ACTION CP03:
{region "CP03柜"}									
DI_[8,1](	ON:= , 	OFF:= , 	LINK:=EL1008[8,1] , 	VALUE=> 	arDropCylinder[11].i.InSensor	);	(*	料仓11气缸原位	*)
DI_[8,2](	ON:= , 	OFF:= , 	LINK:=EL1008[8,2] , 	VALUE=> 	arDropCylinder[11].i.OutSensor	);	(*	料仓11气缸工作位	*)
DI_[8,3](	ON:= , 	OFF:= , 	LINK:=EL1008[8,3] , 	VALUE=> 	arHighSensor[11].i.Link	);	(*	料仓11少料	*)
DI_[8,4](	ON:= , 	OFF:= , 	LINK:=EL1008[8,4] , 	VALUE=> 	arLowSensor[11].i.Link	);	(*	料仓11缺料	*)
DI_[8,5](	ON:= , 	OFF:= , 	LINK:=EL1008[8,5] , 	VALUE=> 	arDropCylinder[12].i.InSensor	);	(*	料仓12气缸原位	*)
DI_[8,6](	ON:= , 	OFF:= , 	LINK:=EL1008[8,6] , 	VALUE=> 	arDropCylinder[12].i.OutSensor	);	(*	料仓12气缸工作位	*)
DI_[8,7](	ON:= , 	OFF:= , 	LINK:=EL1008[8,7] , 	VALUE=> 	arHighSensor[12].i.Link	);	(*	料仓12少料	*)
DI_[8,8](	ON:= , 	OFF:= , 	LINK:=EL1008[8,8] , 	VALUE=> 	arLowSensor[12].i.Link	);	(*	料仓12缺料	*)
DI_[9,1](	ON:= , 	OFF:= , 	LINK:=EL1008[9,1] , 	VALUE=> 	arDropCylinder[13].i.InSensor	);	(*	料仓13气缸原位	*)
DI_[9,2](	ON:= , 	OFF:= , 	LINK:=EL1008[9,2] , 	VALUE=> 	arDropCylinder[13].i.OutSensor	);	(*	料仓13气缸工作位	*)
DI_[9,3](	ON:= , 	OFF:= , 	LINK:=EL1008[9,3] , 	VALUE=> 	arHighSensor[13].i.Link	);	(*	料仓13少料	*)
DI_[9,4](	ON:= , 	OFF:= , 	LINK:=EL1008[9,4] , 	VALUE=> 	arLowSensor[13].i.Link	);	(*	料仓13缺料	*)
DI_[9,5](	ON:= , 	OFF:= , 	LINK:=EL1008[9,5] , 	VALUE=> 	arDropCylinder[14].i.InSensor	);	(*	料仓14气缸原位	*)
DI_[9,6](	ON:= , 	OFF:= , 	LINK:=EL1008[9,6] , 	VALUE=> 	arDropCylinder[14].i.OutSensor	);	(*	料仓14气缸工作位	*)
DI_[9,7](	ON:= , 	OFF:= , 	LINK:=EL1008[9,7] , 	VALUE=> 	arHighSensor[14].i.Link	);	(*	料仓14少料	*)
DI_[9,8](	ON:= , 	OFF:= , 	LINK:=EL1008[9,8] , 	VALUE=> 	arLowSensor[14].i.Link	);	(*	料仓14缺料	*)
DI_[10,1](	ON:= , 	OFF:= , 	LINK:=EL1008[10,1] , 	VALUE=> 	arDropCylinder[15].i.InSensor	);	(*	料仓15气缸原位	*)
DI_[10,2](	ON:= , 	OFF:= , 	LINK:=EL1008[10,2] , 	VALUE=> 	arDropCylinder[15].i.OutSensor	);	(*	料仓15气缸工作位	*)
DI_[10,3](	ON:= , 	OFF:= , 	LINK:=EL1008[10,3] , 	VALUE=> 	arHighSensor[15].i.Link	);	(*	料仓15少料	*)
DI_[10,4](	ON:= , 	OFF:= , 	LINK:=EL1008[10,4] , 	VALUE=> 	arLowSensor[15].i.Link	);	(*	料仓15缺料	*)
DI_[10,5](	ON:= , 	OFF:= , 	LINK:=EL1008[10,5] , 	VALUE=> 	arDropCylinder[16].i.InSensor	);	(*	料仓16气缸原位	*)
DI_[10,6](	ON:= , 	OFF:= , 	LINK:=EL1008[10,6] , 	VALUE=> 	arDropCylinder[16].i.OutSensor	);	(*	料仓16气缸工作位	*)
DI_[10,7](	ON:= , 	OFF:= , 	LINK:=EL1008[10,7] , 	VALUE=> 	arHighSensor[16].i.Link	);	(*	料仓16少料	*)
DI_[10,8](	ON:= , 	OFF:= , 	LINK:=EL1008[10,8] , 	VALUE=> 	arLowSensor[16].i.Link	);	(*	料仓16缺料	*)
DI_[11,1](	ON:= , 	OFF:= , 	LINK:=EL1008[11,1] , 	VALUE=> 	arDropCylinder[17].i.InSensor	);	(*	料仓17气缸原位	*)
DI_[11,2](	ON:= , 	OFF:= , 	LINK:=EL1008[11,2] , 	VALUE=> 	arDropCylinder[17].i.OutSensor	);	(*	料仓17气缸工作位	*)
DI_[11,3](	ON:= , 	OFF:= , 	LINK:=EL1008[11,3] , 	VALUE=> 	arHighSensor[17].i.Link	);	(*	料仓17少料	*)
DI_[11,4](	ON:= , 	OFF:= , 	LINK:=EL1008[11,4] , 	VALUE=> 	arLowSensor[17].i.Link	);	(*	料仓17缺料	*)
DI_[11,5](	ON:= , 	OFF:= , 	LINK:=EL1008[11,5] , 	VALUE=> 	arDropCylinder[18].i.InSensor	);	(*	料仓18气缸原位	*)
DI_[11,6](	ON:= , 	OFF:= , 	LINK:=EL1008[11,6] , 	VALUE=> 	arDropCylinder[18].i.OutSensor	);	(*	料仓18气缸工作位	*)
DI_[11,7](	ON:= , 	OFF:= , 	LINK:=EL1008[11,7] , 	VALUE=> 	arHighSensor[18].i.Link	);	(*	料仓18少料	*)
DI_[11,8](	ON:= , 	OFF:= , 	LINK:=EL1008[11,8] , 	VALUE=> 	arLowSensor[18].i.Link	);	(*	料仓18缺料	*)
DI_[12,1](	ON:= , 	OFF:= , 	LINK:=EL1008[12,1] , 	VALUE=> 	arDropCylinder[19].i.InSensor	);	(*	料仓19气缸原位	*)
DI_[12,2](	ON:= , 	OFF:= , 	LINK:=EL1008[12,2] , 	VALUE=> 	arDropCylinder[19].i.OutSensor	);	(*	料仓19气缸工作位	*)
DI_[12,3](	ON:= , 	OFF:= , 	LINK:=EL1008[12,3] , 	VALUE=> 	arHighSensor[19].i.Link	);	(*	料仓19少料	*)
DI_[12,4](	ON:= , 	OFF:= , 	LINK:=EL1008[12,4] , 	VALUE=> 	arLowSensor[19].i.Link	);	(*	料仓19缺料	*)
DI_[12,5](	ON:= , 	OFF:= , 	LINK:=EL1008[12,5] , 	VALUE=> 	arDropCylinder[20].i.InSensor	);	(*	料仓20气缸原位	*)
DI_[12,6](	ON:= , 	OFF:= , 	LINK:=EL1008[12,6] , 	VALUE=> 	arDropCylinder[20].i.OutSensor	);	(*	料仓20气缸工作位	*)
DI_[12,7](	ON:= , 	OFF:= , 	LINK:=EL1008[12,7] , 	VALUE=> 	arHighSensor[20].i.Link	);	(*	料仓20少料	*)
DI_[12,8](	ON:= , 	OFF:= , 	LINK:=EL1008[12,8] , 	VALUE=> 	arLowSensor[20].i.Link	);	(*	料仓20缺料	*)		
DI_[13,1](	ON:= , 	OFF:= , 	LINK:=EL1008[13,1] , 	VALUE=> 	arDropSensor[11].i.Link	);	(*	工位11落料	*)
DI_[13,2](	ON:= , 	OFF:= , 	LINK:=EL1008[13,2] , 	VALUE=> 	arDropSensor[12].i.Link	);	(*	工位12落料	*)
DI_[13,3](	ON:= , 	OFF:= , 	LINK:=EL1008[13,3] , 	VALUE=> 	arDropSensor[13].i.Link	);	(*	工位13落料	*)
DI_[13,4](	ON:= , 	OFF:= , 	LINK:=EL1008[13,4] , 	VALUE=> 	arDropSensor[14].i.Link	);	(*	工位14落料	*)
DI_[13,5](	ON:= , 	OFF:= , 	LINK:=EL1008[13,5] , 	VALUE=> 	arDropSensor[15].i.Link	);	(*	工位15落料	*)
DI_[13,6](	ON:= , 	OFF:= , 	LINK:=EL1008[13,6] , 	VALUE=> 	arDropSensor[16].i.Link	);	(*	工位16落料	*)
DI_[13,7](	ON:= , 	OFF:= , 	LINK:=EL1008[13,7] , 	VALUE=> 	arDropSensor[17].i.Link	);	(*	工位17落料	*)
DI_[13,8](	ON:= , 	OFF:= , 	LINK:=EL1008[13,8] , 	VALUE=> 	arDropSensor[18].i.Link	);	(*	工位18落料	*)
DI_[14,1](	ON:= , 	OFF:= , 	LINK:=EL1008[14,1] , 	VALUE=> 	arDropSensor[19].i.Link	);	(*	工位19落料	*)
DI_[14,2](	ON:= , 	OFF:= , 	LINK:=EL1008[14,2] , 	VALUE=> 	arDropSensor[20].i.Link	);	(*	工位20落料	*)
DI_[14,3](	ON:= , 	OFF:= , 	LINK:=EL1008[14,3] , 	VALUE=> 	arSafeDoorSts[5]	);	(*	安全门5	*)
DI_[14,4](	ON:= , 	OFF:= , 	LINK:=EL1008[14,4] , 	VALUE=> 	arSafeDoorSts[6]	);	(*	安全门6	*)
DI_[14,5](	ON:= , 	OFF:= , 	LINK:=EL1008[14,5] , 	VALUE=> 	arSafeDoorSts[7]	);	(*	安全门7	*)
DI_[14,6](	ON:= , 	OFF:= , 	LINK:=EL1008[14,6] , 	VALUE=> 	arSafeDoorSts[8]	);	(*	安全门8	*)
DI_[14,7](	ON:= , 	OFF:= , 	LINK:=EL1008[14,7] , 	VALUE=> 	arSafeDoorSts[9]	);	(*	安全门9	*)
DI_[14,8](	ON:= , 	OFF:= , 	LINK:=EL1008[14,8] , 	VALUE=> 	glb_bAirFeedback_UN01[2]	);	(*	数粒系统气压反馈	*)
DI_[30,1](	ON:= , 	OFF:= , 	LINK:=EL1008[30,1] , 	VALUE=> 	arDropBufferCyclinder[1].i.InSensor	);	(*	备用	*)
DI_[30,2](	ON:= , 	OFF:= , 	LINK:=EL1008[30,2] , 	VALUE=> 		);	(*	备用	*)
DI_[30,3](	ON:= , 	OFF:= , 	LINK:=EL1008[30,3] , 	VALUE=> 		);	(*	备用	*)
DI_[30,4](	ON:= , 	OFF:= , 	LINK:=EL1008[30,4] , 	VALUE=> 		);	(*	备用	*)
DI_[30,5](	ON:= , 	OFF:= , 	LINK:=EL1008[30,5] , 	VALUE=> 		);	(*	备用	*)
DI_[30,6](	ON:= , 	OFF:= , 	LINK:=EL1008[30,6] , 	VALUE=> 		);	(*	备用	*)
DI_[30,7](	ON:= , 	OFF:= , 	LINK:=EL1008[30,7] , 	VALUE=> 		);	(*	备用	*)
DI_[30,8](	ON:= , 	OFF:= , 	LINK:=EL1008[30,8] , 	VALUE=> 		);	(*	备用	*)


arDropBufferCyclinder[1].i.OutSensor:= NOT arDropBufferCyclinder[1].i.InSensor;
arDropBufferCyclinder[2].i.OutSensor:= NOT arDropBufferCyclinder[2].i.InSensor;		  
(*****************************************************************************************************)									
DO_[8,1](	ON:= , 	OFF:= , 	LINK=>EL2008[8,1] , 	VALUE:= 	arDropCylinder[11].o.ValveIn	);	(*	料仓11气缸原位	*)
DO_[8,2](	ON:= , 	OFF:= , 	LINK=>EL2008[8,2] , 	VALUE:= 	arDropCylinder[11].o.ValveOut	);	(*	料仓11气缸工作位	*)
DO_[8,3](	ON:= , 	OFF:= , 	LINK=>EL2008[8,3] , 	VALUE:= 	arDropCylinder[12].o.ValveIn	);	(*	料仓12气缸原位	*)
DO_[8,4](	ON:= , 	OFF:= , 	LINK=>EL2008[8,4] , 	VALUE:= 	arDropCylinder[12].o.ValveOut	);	(*	料仓12气缸工作位	*)
DO_[8,5](	ON:= , 	OFF:= , 	LINK=>EL2008[8,5] , 	VALUE:= 	arDropCylinder[13].o.ValveIn	);	(*	料仓13气缸原位	*)
DO_[8,6](	ON:= , 	OFF:= , 	LINK=>EL2008[8,6] , 	VALUE:= 	arDropCylinder[13].o.ValveOut	);	(*	料仓13气缸工作位	*)
DO_[8,7](	ON:= , 	OFF:= , 	LINK=>EL2008[8,7] , 	VALUE:= 	arDropCylinder[14].o.ValveIn	);	(*	料仓14气缸原位	*)
DO_[8,8](	ON:= , 	OFF:= , 	LINK=>EL2008[8,8] , 	VALUE:= 	arDropCylinder[14].o.ValveOut	);	(*	料仓14气缸工作位	*)
DO_[9,1](	ON:= , 	OFF:= , 	LINK=>EL2008[9,1] , 	VALUE:= 	arDropCylinder[15].o.ValveIn	);	(*	料仓15气缸原位	*)
DO_[9,2](	ON:= , 	OFF:= , 	LINK=>EL2008[9,2] , 	VALUE:= 	arDropCylinder[15].o.ValveOut	);	(*	料仓15气缸工作位	*)
DO_[9,3](	ON:= , 	OFF:= , 	LINK=>EL2008[9,3] , 	VALUE:= 	arDropCylinder[16].o.ValveIn	);	(*	料仓16气缸原位	*)
DO_[9,4](	ON:= , 	OFF:= , 	LINK=>EL2008[9,4] , 	VALUE:= 	arDropCylinder[16].o.ValveOut	);	(*	料仓16气缸工作位	*)
DO_[9,5](	ON:= , 	OFF:= , 	LINK=>EL2008[9,5] , 	VALUE:= 	arDropCylinder[17].o.ValveIn	);	(*	料仓17气缸原位	*)
DO_[9,6](	ON:= , 	OFF:= , 	LINK=>EL2008[9,6] , 	VALUE:= 	arDropCylinder[17].o.ValveOut	);	(*	料仓17气缸工作位	*)
DO_[9,7](	ON:= , 	OFF:= , 	LINK=>EL2008[9,7] , 	VALUE:= 	arDropCylinder[18].o.ValveIn	);	(*	料仓18气缸原位	*)
DO_[9,8](	ON:= , 	OFF:= , 	LINK=>EL2008[9,8] , 	VALUE:= 	arDropCylinder[18].o.ValveOut	);	(*	料仓18气缸工作位	*)
DO_[10,1](	ON:= , 	OFF:= , 	LINK=>EL2008[10,1] , 	VALUE:= 	arDropCylinder[19].o.ValveIn	);	(*	料仓19气缸原位	*)
DO_[10,2](	ON:= , 	OFF:= , 	LINK=>EL2008[10,2] , 	VALUE:= 	arDropCylinder[19].o.ValveOut	);	(*	料仓19气缸工作位	*)
DO_[10,3](	ON:= , 	OFF:= , 	LINK=>EL2008[10,3] , 	VALUE:= 	arDropCylinder[20].o.ValveIn	);	(*	料仓20气缸原位	*)
DO_[10,4](	ON:= , 	OFF:= , 	LINK=>EL2008[10,4] , 	VALUE:= 	arDropCylinder[20].o.ValveOut	);	(*	料仓20气缸工作位	*)
DO_[10,5](	ON:= , 	OFF:= , 	LINK=>EL2008[10,5] , 	VALUE:= 	arCounters[11].LineVibrator_Wrk	);	(*	料仓11直震启动	*)
DO_[10,6](	ON:= , 	OFF:= , 	LINK=>EL2008[10,6] , 	VALUE:= 	arCounters[11].CircleVibrator_Wrk	);	(*	料仓11圆震启动	*)
DO_[10,7](	ON:= , 	OFF:= , 	LINK=>EL2008[10,7] , 	VALUE:= 	arCounters[11].DropVibrator_Wrk	);	(*	料仓11落料启动	*)
DO_[10,8](	ON:= , 	OFF:= , 	LINK=>EL2008[10,8] , 	VALUE:= 	arCounters[12].LineVibrator_Wrk	);	(*	料仓12直震启动	*)
DO_[11,1](	ON:= , 	OFF:= , 	LINK=>EL2008[11,1] , 	VALUE:= 	arCounters[12].CircleVibrator_Wrk	);	(*	料仓12圆震启动	*)
DO_[11,2](	ON:= , 	OFF:= , 	LINK=>EL2008[11,2] , 	VALUE:= 	arCounters[12].DropVibrator_Wrk	);	(*	料仓12落料启动	*)
DO_[11,3](	ON:= , 	OFF:= , 	LINK=>EL2008[11,3] , 	VALUE:= 	arCounters[13].LineVibrator_Wrk	);	(*	料仓13直震启动	*)
DO_[11,4](	ON:= , 	OFF:= , 	LINK=>EL2008[11,4] , 	VALUE:= 	arCounters[13].CircleVibrator_Wrk	);	(*	料仓13圆震启动	*)
DO_[11,5](	ON:= , 	OFF:= , 	LINK=>EL2008[11,5] , 	VALUE:= 	arCounters[13].DropVibrator_Wrk	);	(*	料仓13落料启动	*)
DO_[11,6](	ON:= , 	OFF:= , 	LINK=>EL2008[11,6] , 	VALUE:= 	arCounters[14].LineVibrator_Wrk	);	(*	料仓14直震启动	*)
DO_[11,7](	ON:= , 	OFF:= , 	LINK=>EL2008[11,7] , 	VALUE:= 	arCounters[14].CircleVibrator_Wrk	);	(*	料仓14圆震启动	*)
DO_[11,8](	ON:= , 	OFF:= , 	LINK=>EL2008[11,8] , 	VALUE:= 	arCounters[14].DropVibrator_Wrk	);	(*	料仓14落料启动	*)
DO_[12,1](	ON:= , 	OFF:= , 	LINK=>EL2008[12,1] , 	VALUE:= 	arCounters[15].LineVibrator_Wrk	);	(*	料仓15直震启动	*)
DO_[12,2](	ON:= , 	OFF:= , 	LINK=>EL2008[12,2] , 	VALUE:= 	arCounters[15].CircleVibrator_Wrk	);	(*	料仓15圆震启动	*)
DO_[12,3](	ON:= , 	OFF:= , 	LINK=>EL2008[12,3] , 	VALUE:= 	arCounters[15].DropVibrator_Wrk	);	(*	料仓15落料启动	*)
DO_[12,4](	ON:= , 	OFF:= , 	LINK=>EL2008[12,4] , 	VALUE:= 	arCounters[16].LineVibrator_Wrk	);	(*	料仓16直震启动	*)
DO_[12,5](	ON:= , 	OFF:= , 	LINK=>EL2008[12,5] , 	VALUE:= 	arCounters[16].CircleVibrator_Wrk	);	(*	料仓16圆震启动	*)
DO_[12,6](	ON:= , 	OFF:= , 	LINK=>EL2008[12,6] , 	VALUE:= 	arCounters[16].DropVibrator_Wrk	);	(*	料仓16落料启动	*)
DO_[12,7](	ON:= , 	OFF:= , 	LINK=>EL2008[12,7] , 	VALUE:= 	arCounters[17].LineVibrator_Wrk	);	(*	料仓17直震启动	*)
DO_[12,8](	ON:= , 	OFF:= , 	LINK=>EL2008[12,8] , 	VALUE:= 	arCounters[17].CircleVibrator_Wrk	);	(*	料仓17圆震启动	*)
DO_[13,1](	ON:= , 	OFF:= , 	LINK=>EL2008[13,1] , 	VALUE:= 	arCounters[17].DropVibrator_Wrk	);	(*	料仓17落料启动	*)
DO_[13,2](	ON:= , 	OFF:= , 	LINK=>EL2008[13,2] , 	VALUE:= 	arCounters[18].LineVibrator_Wrk	);	(*	料仓18直震启动	*)
DO_[13,3](	ON:= , 	OFF:= , 	LINK=>EL2008[13,3] , 	VALUE:= 	arCounters[18].CircleVibrator_Wrk	);	(*	料仓18圆震启动	*)
DO_[13,4](	ON:= , 	OFF:= , 	LINK=>EL2008[13,4] , 	VALUE:= 	arCounters[18].DropVibrator_Wrk	);	(*	料仓18落料启动	*)
DO_[13,5](	ON:= , 	OFF:= , 	LINK=>EL2008[13,5] , 	VALUE:= 	arCounters[19].LineVibrator_Wrk	);	(*	料仓19直震启动	*)
DO_[13,6](	ON:= , 	OFF:= , 	LINK=>EL2008[13,6] , 	VALUE:= 	arCounters[19].CircleVibrator_Wrk	);	(*	料仓19圆震启动	*)
DO_[13,7](	ON:= , 	OFF:= , 	LINK=>EL2008[13,7] , 	VALUE:= 	arCounters[19].DropVibrator_Wrk	);	(*	料仓19落料启动	*)
DO_[13,8](	ON:= , 	OFF:= , 	LINK=>EL2008[13,8] , 	VALUE:= 	arCounters[20].LineVibrator_Wrk	);	(*	料仓20直震启动	*)
DO_[14,1](	ON:= , 	OFF:= , 	LINK=>EL2008[14,1] , 	VALUE:= 	arCounters[20].CircleVibrator_Wrk	);	(*	料仓20圆震启动	*)
DO_[14,2](	ON:= , 	OFF:= , 	LINK=>EL2008[14,2] , 	VALUE:= 	arCounters[20].DropVibrator_Wrk	);	(*	料仓20落料启动	*)
DO_[14,3](	ON:= , 	OFF:= , 	LINK=>EL2008[14,3] , 	VALUE:= 	glb_arLightRelay_UN01[1]	);	(*设备照明灯继电器1	*)
DO_[14,4](	ON:= , 	OFF:= , 	LINK=>EL2008[14,4] , 	VALUE:= 	glb_bCounterAirValve_UN01	);	(*数粒系统气压阀	*)
DO_[14,5](	ON:= , 	OFF:= , 	LINK=>EL2008[14,5] , 	VALUE:=     arDropBufferCyclinder[1].o.ValveOut);	(**)
DO_[14,6](	ON:= , 	OFF:= , 	LINK=>EL2008[14,6] , 	VALUE:= 	arDropBufferCyclinder[2].o.ValveOut);	(**)
DO_[14,7](	ON:= , 	OFF:= , 	LINK=>EL2008[14,7] , 	VALUE:= 	);	(**)
DO_[14,8](	ON:= , 	OFF:= , 	LINK=>EL2008[14,8] , 	VALUE:= 	);	(**)									
{endregion}
END_ACTION

ACTION CP04:
{region "CP04柜"}									
DI_[15,1](	ON:= , 	OFF:= , 	LINK:=EL1008[15,1] , 	VALUE=> 	arDropCylinder[21].i.InSensor	);	(*	料仓21气缸原位	*)
DI_[15,2](	ON:= , 	OFF:= , 	LINK:=EL1008[15,2] , 	VALUE=> 	arDropCylinder[21].i.OutSensor	);	(*	料仓21气缸工作位	*)
DI_[15,3](	ON:= , 	OFF:= , 	LINK:=EL1008[15,3] , 	VALUE=> 	arHighSensor[21].i.Link	);	(*	料仓21少料	*)
DI_[15,4](	ON:= , 	OFF:= , 	LINK:=EL1008[15,4] , 	VALUE=> 	arLowSensor[21].i.Link	);	(*	料仓21缺料	*)
DI_[15,5](	ON:= , 	OFF:= , 	LINK:=EL1008[15,5] , 	VALUE=> 	arDropCylinder[22].i.InSensor	);	(*	料仓22气缸原位	*)
DI_[15,6](	ON:= , 	OFF:= , 	LINK:=EL1008[15,6] , 	VALUE=> 	arDropCylinder[22].i.OutSensor	);	(*	料仓22气缸工作位	*)
DI_[15,7](	ON:= , 	OFF:= , 	LINK:=EL1008[15,7] , 	VALUE=> 	arHighSensor[22].i.Link	);	(*	料仓22少料	*)
DI_[15,8](	ON:= , 	OFF:= , 	LINK:=EL1008[15,8] , 	VALUE=> 	arLowSensor[22].i.Link	);	(*	料仓22缺料	*)
DI_[16,1](	ON:= , 	OFF:= , 	LINK:=EL1008[16,1] , 	VALUE=> 	arDropCylinder[23].i.InSensor	);	(*	料仓23气缸原位	*)
DI_[16,2](	ON:= , 	OFF:= , 	LINK:=EL1008[16,2] , 	VALUE=> 	arDropCylinder[23].i.OutSensor	);	(*	料仓23气缸工作位	*)
DI_[16,3](	ON:= , 	OFF:= , 	LINK:=EL1008[16,3] , 	VALUE=> 	arHighSensor[23].i.Link	);	(*	料仓23少料	*)
DI_[16,4](	ON:= , 	OFF:= , 	LINK:=EL1008[16,4] , 	VALUE=> 	arLowSensor[23].i.Link	);	(*	料仓23缺料	*)
DI_[16,5](	ON:= , 	OFF:= , 	LINK:=EL1008[16,5] , 	VALUE=> 	arDropCylinder[24].i.InSensor	);	(*	料仓24气缸原位	*)
DI_[16,6](	ON:= , 	OFF:= , 	LINK:=EL1008[16,6] , 	VALUE=> 	arDropCylinder[24].i.OutSensor	);	(*	料仓24气缸工作位	*)
DI_[16,7](	ON:= , 	OFF:= , 	LINK:=EL1008[16,7] , 	VALUE=> 	arHighSensor[24].i.Link	);	(*	料仓24少料	*)
DI_[16,8](	ON:= , 	OFF:= , 	LINK:=EL1008[16,8] , 	VALUE=> 	arLowSensor[24].i.Link	);	(*	料仓24缺料	*)
DI_[17,1](	ON:= , 	OFF:= , 	LINK:=EL1008[17,1] , 	VALUE=> 	arDropCylinder[25].i.InSensor	);	(*	料仓25气缸原位	*)
DI_[17,2](	ON:= , 	OFF:= , 	LINK:=EL1008[17,2] , 	VALUE=> 	arDropCylinder[25].i.OutSensor	);	(*	料仓25气缸工作位	*)
DI_[17,3](	ON:= , 	OFF:= , 	LINK:=EL1008[17,3] , 	VALUE=> 	arHighSensor[25].i.Link	);	(*	料仓25少料	*)
DI_[17,4](	ON:= , 	OFF:= , 	LINK:=EL1008[17,4] , 	VALUE=> 	arLowSensor[25].i.Link	);	(*	料仓25缺料	*)
DI_[17,5](	ON:= , 	OFF:= , 	LINK:=EL1008[17,5] , 	VALUE=> 	arDropCylinder[26].i.InSensor	);	(*	料仓26气缸原位	*)
DI_[17,6](	ON:= , 	OFF:= , 	LINK:=EL1008[17,6] , 	VALUE=> 	arDropCylinder[26].i.OutSensor	);	(*	料仓26气缸工作位	*)
DI_[17,7](	ON:= , 	OFF:= , 	LINK:=EL1008[17,7] , 	VALUE=> 	arHighSensor[26].i.Link	);	(*	料仓26少料	*)
DI_[17,8](	ON:= , 	OFF:= , 	LINK:=EL1008[17,8] , 	VALUE=> 	arLowSensor[26].i.Link	);	(*	料仓26缺料	*)
DI_[18,1](	ON:= , 	OFF:= , 	LINK:=EL1008[18,1] , 	VALUE=> 	arDropCylinder[27].i.InSensor	);	(*	料仓27气缸原位	*)
DI_[18,2](	ON:= , 	OFF:= , 	LINK:=EL1008[18,2] , 	VALUE=> 	arDropCylinder[27].i.OutSensor	);	(*	料仓27气缸工作位	*)
DI_[18,3](	ON:= , 	OFF:= , 	LINK:=EL1008[18,3] , 	VALUE=> 	arHighSensor[27].i.Link	);	(*	料仓27少料	*)
DI_[18,4](	ON:= , 	OFF:= , 	LINK:=EL1008[18,4] , 	VALUE=> 	arLowSensor[27].i.Link	);	(*	料仓27缺料	*)
DI_[18,5](	ON:= , 	OFF:= , 	LINK:=EL1008[18,5] , 	VALUE=> 	arDropCylinder[28].i.InSensor	);	(*	料仓28气缸原位	*)
DI_[18,6](	ON:= , 	OFF:= , 	LINK:=EL1008[18,6] , 	VALUE=> 	arDropCylinder[28].i.OutSensor	);	(*	料仓28气缸工作位	*)
DI_[18,7](	ON:= , 	OFF:= , 	LINK:=EL1008[18,7] , 	VALUE=> 	arHighSensor[28].i.Link	);	(*	料仓28少料	*)
DI_[18,8](	ON:= , 	OFF:= , 	LINK:=EL1008[18,8] , 	VALUE=> 	arLowSensor[28].i.Link	);	(*	料仓28缺料	*)
DI_[19,1](	ON:= , 	OFF:= , 	LINK:=EL1008[19,1] , 	VALUE=> 	arDropCylinder[29].i.InSensor	);	(*	料仓29气缸原位	*)
DI_[19,2](	ON:= , 	OFF:= , 	LINK:=EL1008[19,2] , 	VALUE=> 	arDropCylinder[29].i.OutSensor	);	(*	料仓29气缸工作位	*)
DI_[19,3](	ON:= , 	OFF:= , 	LINK:=EL1008[19,3] , 	VALUE=> 	arHighSensor[29].i.Link	);	(*	料仓29少料	*)
DI_[19,4](	ON:= , 	OFF:= , 	LINK:=EL1008[19,4] , 	VALUE=> 	arLowSensor[29].i.Link	);	(*	料仓29缺料	*)
DI_[19,5](	ON:= , 	OFF:= , 	LINK:=EL1008[19,5] , 	VALUE=> 	arDropCylinder[30].i.InSensor	);	(*	料仓30气缸原位	*)
DI_[19,6](	ON:= , 	OFF:= , 	LINK:=EL1008[19,6] , 	VALUE=> 	arDropCylinder[30].i.OutSensor	);	(*	料仓30气缸工作位	*)
DI_[19,7](	ON:= , 	OFF:= , 	LINK:=EL1008[19,7] , 	VALUE=> 	arHighSensor[30].i.Link	);	(*	料仓30少料	*)
DI_[19,8](	ON:= , 	OFF:= , 	LINK:=EL1008[19,8] , 	VALUE=> 	arLowSensor[30].i.Link	);	(*	料仓30缺料	*)
DI_[20,1](	ON:= , 	OFF:= , 	LINK:=EL1008[20,1] , 	VALUE=> 	arDropSensor[21].i.Link	);	(*	工位21落料	*)
DI_[20,2](	ON:= , 	OFF:= , 	LINK:=EL1008[20,2] , 	VALUE=> 	arDropSensor[22].i.Link	);	(*	工位22落料	*)
DI_[20,3](	ON:= , 	OFF:= , 	LINK:=EL1008[20,3] , 	VALUE=> 	arDropSensor[23].i.Link	);	(*	工位23落料	*)
DI_[20,4](	ON:= , 	OFF:= , 	LINK:=EL1008[20,4] , 	VALUE=> 	arDropSensor[24].i.Link	);	(*	工位24落料	*)
DI_[20,5](	ON:= , 	OFF:= , 	LINK:=EL1008[20,5] , 	VALUE=> 	arDropSensor[25].i.Link	);	(*	工位25落料	*)
DI_[20,6](	ON:= , 	OFF:= , 	LINK:=EL1008[20,6] , 	VALUE=> 	arDropSensor[26].i.Link	);	(*	工位26落料	*)
DI_[20,7](	ON:= , 	OFF:= , 	LINK:=EL1008[20,7] , 	VALUE=> 	arDropSensor[27].i.Link	);	(*	工位27落料	*)
DI_[20,8](	ON:= , 	OFF:= , 	LINK:=EL1008[20,8] , 	VALUE=> 	arDropSensor[28].i.Link	);	(*	工位28落料	*)
DI_[21,1](	ON:= , 	OFF:= , 	LINK:=EL1008[21,1] , 	VALUE=> 	arDropSensor[29].i.Link	);	(*	工位29落料	*)
DI_[21,2](	ON:= , 	OFF:= , 	LINK:=EL1008[21,2] , 	VALUE=> 	arDropSensor[30].i.Link	);	(*	工位30落料	*)
DI_[21,3](	ON:= , 	OFF:= , 	LINK:=EL1008[21,3] , 	VALUE=> 	arSafeDoorSts[10]	);	(*	安全门10	*)
DI_[21,4](	ON:= , 	OFF:= , 	LINK:=EL1008[21,4] , 	VALUE=> 	arSafeDoorSts[11]	);	(*	安全门11	*)
DI_[21,5](	ON:= , 	OFF:= , 	LINK:=EL1008[21,5] , 	VALUE=> 	arSafeDoorSts[12]	);	(*	安全门12	*)
DI_[21,6](	ON:= , 	OFF:= , 	LINK:=EL1008[21,6] , 	VALUE=> 	arSafeDoorSts[13]	);	(*	安全门13	*)
DI_[21,7](	ON:= , 	OFF:= , 	LINK:=EL1008[21,7] , 	VALUE=> 	arSafeDoorSts[14]	);	(*	安全门14	*)
DI_[21,8](	ON:= , 	OFF:= , 	LINK:=EL1008[21,8] , 	VALUE=> 		);	(*	预留急停反馈*)
DI_[31,1](	ON:= , 	OFF:= , 	LINK:=EL1008[31,1] , 	VALUE=> 		);	(*	备用	*)
DI_[31,2](	ON:= , 	OFF:= , 	LINK:=EL1008[31,2] , 	VALUE=> 		);	(*	备用	*)
DI_[31,3](	ON:= , 	OFF:= , 	LINK:=EL1008[31,3] , 	VALUE=> 		);	(*	备用	*)
DI_[31,4](	ON:= , 	OFF:= , 	LINK:=EL1008[31,4] , 	VALUE=> 		);	(*	备用	*)
DI_[31,5](	ON:= , 	OFF:= , 	LINK:=EL1008[31,5] , 	VALUE=> 		);	(*	备用	*)
DI_[31,6](	ON:= , 	OFF:= , 	LINK:=EL1008[31,6] , 	VALUE=> 		);	(*	备用	*)
DI_[31,7](	ON:= , 	OFF:= , 	LINK:=EL1008[31,7] , 	VALUE=> 		);	(*	备用	*)
DI_[31,8](	ON:= , 	OFF:= , 	LINK:=EL1008[31,8] , 	VALUE=> 		);	(*	备用	*)

	 
		  
			   
					
						 
							  
								   
(*****************************************************************************************************)									
DO_[15,1](	ON:= , 	OFF:= , 	LINK=>EL2008[15,1] , 	VALUE:= 	arDropCylinder[21].o.ValveIn	);	(*	料仓21气缸原位	*)
DO_[15,2](	ON:= , 	OFF:= , 	LINK=>EL2008[15,2] , 	VALUE:= 	arDropCylinder[21].o.ValveOut	);	(*	料仓21气缸工作位	*)
DO_[15,3](	ON:= , 	OFF:= , 	LINK=>EL2008[15,3] , 	VALUE:= 	arDropCylinder[22].o.ValveIn	);	(*	料仓22气缸原位	*)
DO_[15,4](	ON:= , 	OFF:= , 	LINK=>EL2008[15,4] , 	VALUE:= 	arDropCylinder[22].o.ValveOut	);	(*	料仓22气缸工作位	*)
DO_[15,5](	ON:= , 	OFF:= , 	LINK=>EL2008[15,5] , 	VALUE:= 	arDropCylinder[23].o.ValveIn	);	(*	料仓23气缸原位	*)
DO_[15,6](	ON:= , 	OFF:= , 	LINK=>EL2008[15,6] , 	VALUE:= 	arDropCylinder[23].o.ValveOut	);	(*	料仓23气缸工作位	*)
DO_[15,7](	ON:= , 	OFF:= , 	LINK=>EL2008[15,7] , 	VALUE:= 	arDropCylinder[24].o.ValveIn	);	(*	料仓24气缸原位	*)
DO_[15,8](	ON:= , 	OFF:= , 	LINK=>EL2008[15,8] , 	VALUE:= 	arDropCylinder[24].o.ValveOut	);	(*	料仓24气缸工作位	*)
DO_[16,1](	ON:= , 	OFF:= , 	LINK=>EL2008[16,1] , 	VALUE:= 	arDropCylinder[25].o.ValveIn	);	(*	料仓25气缸原位	*)
DO_[16,2](	ON:= , 	OFF:= , 	LINK=>EL2008[16,2] , 	VALUE:= 	arDropCylinder[25].o.ValveOut	);	(*	料仓25气缸工作位	*)
DO_[16,3](	ON:= , 	OFF:= , 	LINK=>EL2008[16,3] , 	VALUE:= 	arDropCylinder[26].o.ValveIn	);	(*	料仓26气缸原位	*)
DO_[16,4](	ON:= , 	OFF:= , 	LINK=>EL2008[16,4] , 	VALUE:= 	arDropCylinder[26].o.ValveOut	);	(*	料仓26气缸工作位	*)
DO_[16,5](	ON:= , 	OFF:= , 	LINK=>EL2008[16,5] , 	VALUE:= 	arDropCylinder[27].o.ValveIn	);	(*	料仓27气缸原位	*)
DO_[16,6](	ON:= , 	OFF:= , 	LINK=>EL2008[16,6] , 	VALUE:= 	arDropCylinder[27].o.ValveOut	);	(*	料仓27气缸工作位	*)
DO_[16,7](	ON:= , 	OFF:= , 	LINK=>EL2008[16,7] , 	VALUE:= 	arDropCylinder[28].o.ValveIn	);	(*	料仓28气缸原位	*)
DO_[16,8](	ON:= , 	OFF:= , 	LINK=>EL2008[16,8] , 	VALUE:= 	arDropCylinder[28].o.ValveOut	);	(*	料仓28气缸工作位	*)
DO_[17,1](	ON:= , 	OFF:= , 	LINK=>EL2008[17,1] , 	VALUE:= 	arDropCylinder[29].o.ValveIn	);	(*	料仓29气缸原位	*)
DO_[17,2](	ON:= , 	OFF:= , 	LINK=>EL2008[17,2] , 	VALUE:= 	arDropCylinder[29].o.ValveOut	);	(*	料仓29气缸工作位	*)
DO_[17,3](	ON:= , 	OFF:= , 	LINK=>EL2008[17,3] , 	VALUE:= 	arDropCylinder[30].o.ValveIn	);	(*	料仓30气缸原位	*)
DO_[17,4](	ON:= , 	OFF:= , 	LINK=>EL2008[17,4] , 	VALUE:= 	arDropCylinder[30].o.ValveOut	);	(*	料仓30气缸工作位	*)
DO_[17,5](	ON:= , 	OFF:= , 	LINK=>EL2008[17,5] , 	VALUE:= 	arCounters[21].LineVibrator_Wrk	);	(*	料仓21直震启动	*)
DO_[17,6](	ON:= , 	OFF:= , 	LINK=>EL2008[17,6] , 	VALUE:= 	arCounters[21].CircleVibrator_Wrk	);	(*	料仓21圆震启动	*)
DO_[17,7](	ON:= , 	OFF:= , 	LINK=>EL2008[17,7] , 	VALUE:= 	arCounters[21].DropVibrator_Wrk	);	(*	料仓21落料启动	*)
DO_[17,8](	ON:= , 	OFF:= , 	LINK=>EL2008[17,8] , 	VALUE:= 	arCounters[22].LineVibrator_Wrk	);	(*	料仓22直震启动	*)
DO_[18,1](	ON:= , 	OFF:= , 	LINK=>EL2008[18,1] , 	VALUE:= 	arCounters[22].CircleVibrator_Wrk	);	(*	料仓22圆震启动	*)
DO_[18,2](	ON:= , 	OFF:= , 	LINK=>EL2008[18,2] , 	VALUE:= 	arCounters[22].DropVibrator_Wrk	);	(*	料仓22落料启动	*)
DO_[18,3](	ON:= , 	OFF:= , 	LINK=>EL2008[18,3] , 	VALUE:= 	arCounters[23].LineVibrator_Wrk	);	(*	料仓23直震启动	*)
DO_[18,4](	ON:= , 	OFF:= , 	LINK=>EL2008[18,4] , 	VALUE:= 	arCounters[23].CircleVibrator_Wrk	);	(*	料仓23圆震启动	*)
DO_[18,5](	ON:= , 	OFF:= , 	LINK=>EL2008[18,5] , 	VALUE:= 	arCounters[23].DropVibrator_Wrk	);	(*	料仓23落料启动	*)
DO_[18,6](	ON:= , 	OFF:= , 	LINK=>EL2008[18,6] , 	VALUE:= 	arCounters[24].LineVibrator_Wrk	);	(*	料仓24直震启动	*)
DO_[18,7](	ON:= , 	OFF:= , 	LINK=>EL2008[18,7] , 	VALUE:= 	arCounters[24].CircleVibrator_Wrk	);	(*	料仓24圆震启动	*)
DO_[18,8](	ON:= , 	OFF:= , 	LINK=>EL2008[18,8] , 	VALUE:= 	arCounters[24].DropVibrator_Wrk	);	(*	料仓24落料启动	*)
DO_[19,1](	ON:= , 	OFF:= , 	LINK=>EL2008[19,1] , 	VALUE:= 	arCounters[25].LineVibrator_Wrk	);	(*	料仓25直震启动	*)
DO_[19,2](	ON:= , 	OFF:= , 	LINK=>EL2008[19,2] , 	VALUE:= 	arCounters[25].CircleVibrator_Wrk	);	(*	料仓25圆震启动	*)
DO_[19,3](	ON:= , 	OFF:= , 	LINK=>EL2008[19,3] , 	VALUE:= 	arCounters[25].DropVibrator_Wrk	);	(*	料仓25落料启动	*)
DO_[19,4](	ON:= , 	OFF:= , 	LINK=>EL2008[19,4] , 	VALUE:= 	arCounters[26].LineVibrator_Wrk	);	(*	料仓26直震启动	*)
DO_[19,5](	ON:= , 	OFF:= , 	LINK=>EL2008[19,5] , 	VALUE:= 	arCounters[26].CircleVibrator_Wrk	);	(*	料仓26圆震启动	*)
DO_[19,6](	ON:= , 	OFF:= , 	LINK=>EL2008[19,6] , 	VALUE:= 	arCounters[26].DropVibrator_Wrk	);	(*	料仓26落料启动	*)
DO_[19,7](	ON:= , 	OFF:= , 	LINK=>EL2008[19,7] , 	VALUE:= 	arCounters[27].LineVibrator_Wrk	);	(*	料仓27直震启动	*)
DO_[19,8](	ON:= , 	OFF:= , 	LINK=>EL2008[19,8] , 	VALUE:= 	arCounters[27].CircleVibrator_Wrk	);	(*	料仓27圆震启动	*)
DO_[20,1](	ON:= , 	OFF:= , 	LINK=>EL2008[20,1] , 	VALUE:= 	arCounters[27].DropVibrator_Wrk	);	(*	料仓27落料启动	*)
DO_[20,2](	ON:= , 	OFF:= , 	LINK=>EL2008[20,2] , 	VALUE:= 	arCounters[28].LineVibrator_Wrk	);	(*	料仓28直震启动	*)
DO_[20,3](	ON:= , 	OFF:= , 	LINK=>EL2008[20,3] , 	VALUE:= 	arCounters[28].CircleVibrator_Wrk	);	(*	料仓28圆震启动	*)
DO_[20,4](	ON:= , 	OFF:= , 	LINK=>EL2008[20,4] , 	VALUE:=     arCounters[28].DropVibrator_Wrk	);	(*	料仓28落料启动	*)
DO_[20,5](	ON:= , 	OFF:= , 	LINK=>EL2008[20,5] , 	VALUE:= 	arCounters[29].LineVibrator_Wrk	);	(*	料仓29直震启动	*)
DO_[20,6](	ON:= , 	OFF:= , 	LINK=>EL2008[20,6] , 	VALUE:= 	arCounters[29].CircleVibrator_Wrk	);	(*	料仓29圆震启动	*)
DO_[20,7](	ON:= , 	OFF:= , 	LINK=>EL2008[20,7] , 	VALUE:= 	arCounters[29].DropVibrator_Wrk	);	(*	料仓29落料启动	*)
DO_[20,8](	ON:= , 	OFF:= , 	LINK=>EL2008[20,8] , 	VALUE:= 	arCounters[30].LineVibrator_Wrk	);	(*	料仓30直震启动	*)
DO_[21,1](	ON:= , 	OFF:= , 	LINK=>EL2008[21,1] , 	VALUE:= 	arCounters[30].CircleVibrator_Wrk	);	(*	料仓30圆震启动	*)
DO_[21,2](	ON:= , 	OFF:= , 	LINK=>EL2008[21,2] , 	VALUE:= 	arCounters[30].DropVibrator_Wrk	);	(*	料仓30落料启动	*)
DO_[21,3](	ON:= , 	OFF:= , 	LINK=>EL2008[21,3] , 	VALUE:= 	glb_arLightRed_UN01[2]	);	(*	备用	*)
DO_[21,4](	ON:= , 	OFF:= , 	LINK=>EL2008[21,4] , 	VALUE:= 	glb_arLightYellow_UN01[2]	);	(*	备用	*)
DO_[21,5](	ON:= , 	OFF:= , 	LINK=>EL2008[21,5] , 	VALUE:= 	glb_arLightGreen_UN01[2]	);	(*	备用	*)
DO_[21,6](	ON:= , 	OFF:= , 	LINK=>EL2008[21,6] , 	VALUE:= 	glb_arLightAlarm_UN01[2]	);	(*	备用	*)
DO_[21,7](	ON:= , 	OFF:= , 	LINK=>EL2008[21,7] , 	VALUE:= 		);	(*	备用	*)
DO_[21,8](	ON:= , 	OFF:= , 	LINK=>EL2008[21,8] , 	VALUE:= 		);	(*	备用	*)
									
{endregion}
END_ACTION

ACTION CP05:
{region "CP05柜"}									
DI_[22,1](	ON:= , 	OFF:= , 	LINK:=EL1008[22,1] , 	VALUE=> 	arDropCylinder[31].i.InSensor	);	(*	料仓31气缸原位	*)
DI_[22,2](	ON:= , 	OFF:= , 	LINK:=EL1008[22,2] , 	VALUE=> 	arDropCylinder[31].i.OutSensor	);	(*	料仓31气缸工作位	*)
DI_[22,3](	ON:= , 	OFF:= , 	LINK:=EL1008[22,3] , 	VALUE=> 	arHighSensor[31].i.Link	);	(*	料仓31少料	*)
DI_[22,4](	ON:= , 	OFF:= , 	LINK:=EL1008[22,4] , 	VALUE=> 	arLowSensor[31].i.Link	);	(*	料仓31缺料	*)
DI_[22,5](	ON:= , 	OFF:= , 	LINK:=EL1008[22,5] , 	VALUE=> 	arDropCylinder[32].i.InSensor	);	(*	料仓32气缸原位	*)
DI_[22,6](	ON:= , 	OFF:= , 	LINK:=EL1008[22,6] , 	VALUE=> 	arDropCylinder[32].i.OutSensor	);	(*	料仓32气缸工作位	*)
DI_[22,7](	ON:= , 	OFF:= , 	LINK:=EL1008[22,7] , 	VALUE=> 	arHighSensor[32].i.Link	);	(*	料仓32少料	*)
DI_[22,8](	ON:= , 	OFF:= , 	LINK:=EL1008[22,8] , 	VALUE=> 	arLowSensor[32].i.Link	);	(*	料仓32缺料	*)
DI_[23,1](	ON:= , 	OFF:= , 	LINK:=EL1008[23,1] , 	VALUE=> 	arDropCylinder[33].i.InSensor	);	(*	料仓33气缸原位	*)
DI_[23,2](	ON:= , 	OFF:= , 	LINK:=EL1008[23,2] , 	VALUE=> 	arDropCylinder[33].i.OutSensor	);	(*	料仓33气缸工作位	*)
DI_[23,3](	ON:= , 	OFF:= , 	LINK:=EL1008[23,3] , 	VALUE=> 	arHighSensor[33].i.Link	);	(*	料仓33少料	*)
DI_[23,4](	ON:= , 	OFF:= , 	LINK:=EL1008[23,4] , 	VALUE=> 	arLowSensor[33].i.Link	);	(*	料仓33缺料	*)
DI_[23,5](	ON:= , 	OFF:= , 	LINK:=EL1008[23,5] , 	VALUE=> 	arDropCylinder[34].i.InSensor	);	(*	料仓34气缸原位	*)
DI_[23,6](	ON:= , 	OFF:= , 	LINK:=EL1008[23,6] , 	VALUE=> 	arDropCylinder[34].i.OutSensor	);	(*	料仓34气缸工作位	*)
DI_[23,7](	ON:= , 	OFF:= , 	LINK:=EL1008[23,7] , 	VALUE=> 	arHighSensor[34].i.Link	);	(*	料仓34少料	*)
DI_[23,8](	ON:= , 	OFF:= , 	LINK:=EL1008[23,8] , 	VALUE=> 	arLowSensor[34].i.Link	);	(*	料仓34缺料	*)
DI_[24,1](	ON:= , 	OFF:= , 	LINK:=EL1008[24,1] , 	VALUE=> 	arDropCylinder[35].i.InSensor	);	(*	料仓35气缸原位	*)
DI_[24,2](	ON:= , 	OFF:= , 	LINK:=EL1008[24,2] , 	VALUE=> 	arDropCylinder[35].i.OutSensor	);	(*	料仓35气缸工作位	*)
DI_[24,3](	ON:= , 	OFF:= , 	LINK:=EL1008[24,3] , 	VALUE=> 	arHighSensor[35].i.Link	);	(*	料仓35少料	*)
DI_[24,4](	ON:= , 	OFF:= , 	LINK:=EL1008[24,4] , 	VALUE=> 	arLowSensor[35].i.Link	);	(*	料仓35缺料	*)
DI_[24,5](	ON:= , 	OFF:= , 	LINK:=EL1008[24,5] , 	VALUE=> 	arDropCylinder[36].i.InSensor	);	(*	料仓36气缸原位	*)
DI_[24,6](	ON:= , 	OFF:= , 	LINK:=EL1008[24,6] , 	VALUE=> 	arDropCylinder[36].i.OutSensor	);	(*	料仓36气缸工作位	*)
DI_[24,7](	ON:= , 	OFF:= , 	LINK:=EL1008[24,7] , 	VALUE=> 	arHighSensor[36].i.Link	);	(*	料仓36少料	*)
DI_[24,8](	ON:= , 	OFF:= , 	LINK:=EL1008[24,8] , 	VALUE=> 	arLowSensor[36].i.Link	);	(*	料仓36缺料	*)
DI_[25,1](	ON:= , 	OFF:= , 	LINK:=EL1008[25,1] , 	VALUE=> 	arDropCylinder[37].i.InSensor	);	(*	料仓37气缸原位	*)
DI_[25,2](	ON:= , 	OFF:= , 	LINK:=EL1008[25,2] , 	VALUE=> 	arDropCylinder[37].i.OutSensor	);	(*	料仓37气缸工作位	*)
DI_[25,3](	ON:= , 	OFF:= , 	LINK:=EL1008[25,3] , 	VALUE=> 	arHighSensor[37].i.Link	);	(*	料仓37少料	*)
DI_[25,4](	ON:= , 	OFF:= , 	LINK:=EL1008[25,4] , 	VALUE=> 	arLowSensor[37].i.Link	);	(*	料仓37缺料	*)
DI_[25,5](	ON:= , 	OFF:= , 	LINK:=EL1008[25,5] , 	VALUE=> 	arDropCylinder[38].i.InSensor	);	(*	料仓38气缸原位	*)
DI_[25,6](	ON:= , 	OFF:= , 	LINK:=EL1008[25,6] , 	VALUE=> 	arDropCylinder[38].i.OutSensor	);	(*	料仓38气缸工作位	*)
DI_[25,7](	ON:= , 	OFF:= , 	LINK:=EL1008[25,7] , 	VALUE=> 	arHighSensor[38].i.Link	);	(*	料仓38少料	*)
DI_[25,8](	ON:= , 	OFF:= , 	LINK:=EL1008[25,8] , 	VALUE=> 	arLowSensor[38].i.Link	);	(*	料仓38缺料	*)
DI_[26,1](	ON:= , 	OFF:= , 	LINK:=EL1008[26,1] , 	VALUE=> 	arDropCylinder[39].i.InSensor	);	(*	料仓39气缸原位	*)
DI_[26,2](	ON:= , 	OFF:= , 	LINK:=EL1008[26,2] , 	VALUE=> 	arDropCylinder[39].i.OutSensor	);	(*	料仓39气缸工作位	*)
DI_[26,3](	ON:= , 	OFF:= , 	LINK:=EL1008[26,3] , 	VALUE=> 	arHighSensor[39].i.Link	);	(*	料仓39少料	*)
DI_[26,4](	ON:= , 	OFF:= , 	LINK:=EL1008[26,4] , 	VALUE=> 	arLowSensor[39].i.Link	);	(*	料仓39缺料	*)
DI_[26,5](	ON:= , 	OFF:= , 	LINK:=EL1008[26,5] , 	VALUE=> 	arDropCylinder[40].i.InSensor	);	(*	料仓40气缸原位	*)
DI_[26,6](	ON:= , 	OFF:= , 	LINK:=EL1008[26,6] , 	VALUE=> 	arDropCylinder[40].i.OutSensor	);	(*	料仓40气缸工作位	*)
DI_[26,7](	ON:= , 	OFF:= , 	LINK:=EL1008[26,7] , 	VALUE=> 	arHighSensor[40].i.Link	);	(*	料仓40少料	*)
DI_[26,8](	ON:= , 	OFF:= , 	LINK:=EL1008[26,8] , 	VALUE=> 	arLowSensor[40].i.Link	);	(*	料仓40缺料	*)
DI_[27,1](	ON:= , 	OFF:= , 	LINK:=EL1008[27,1] , 	VALUE=> 	arDropSensor[31].i.Link	);	(*	工位31落料	*)
DI_[27,2](	ON:= , 	OFF:= , 	LINK:=EL1008[27,2] , 	VALUE=> 	arDropSensor[32].i.Link	);	(*	工位32落料	*)
DI_[27,3](	ON:= , 	OFF:= , 	LINK:=EL1008[27,3] , 	VALUE=> 	arDropSensor[33].i.Link	);	(*	工位33落料	*)
DI_[27,4](	ON:= , 	OFF:= , 	LINK:=EL1008[27,4] , 	VALUE=> 	arDropSensor[34].i.Link	);	(*	工位34落料	*)
DI_[27,5](	ON:= , 	OFF:= , 	LINK:=EL1008[27,5] , 	VALUE=> 	arDropSensor[35].i.Link	);	(*	工位35落料	*)
DI_[27,6](	ON:= , 	OFF:= , 	LINK:=EL1008[27,6] , 	VALUE=> 	arDropSensor[36].i.Link	);	(*	工位36落料	*)
DI_[27,7](	ON:= , 	OFF:= , 	LINK:=EL1008[27,7] , 	VALUE=> 	arDropSensor[37].i.Link	);	(*	工位37落料	*)
DI_[27,1](	ON:= , 	OFF:= , 	LINK:=EL1008[27,8] , 	VALUE=> 	arDropSensor[38].i.Link	);	(*	工位38落料	*)
DI_[28,1](	ON:= , 	OFF:= , 	LINK:=EL1008[28,1] , 	VALUE=> 	arDropSensor[39].i.Link	);	(*	工位39落料	*)
DI_[28,2](	ON:= , 	OFF:= , 	LINK:=EL1008[28,2] , 	VALUE=> 	arDropSensor[40].i.Link	);	(*	工位40落料	*)
DI_[28,3](	ON:= , 	OFF:= , 	LINK:=EL1008[28,3] , 	VALUE=> 	arSafeDoorSts[15]	);	(*	安全门15	*)
DI_[28,4](	ON:= , 	OFF:= , 	LINK:=EL1008[28,4] , 	VALUE=> 	arSafeDoorSts[16]	);	(*	安全门16	*)
DI_[28,5](	ON:= , 	OFF:= , 	LINK:=EL1008[28,5] , 	VALUE=> 	arSafeDoorSts[17]	);	(*	安全门17	*)
DI_[28,6](	ON:= , 	OFF:= , 	LINK:=EL1008[28,6] , 	VALUE=> 	arSafeDoorSts[18]	);	(*	安全门18	*)
DI_[28,7](	ON:= , 	OFF:= , 	LINK:=EL1008[28,7] , 	VALUE=> 		);	(*		*)
DI_[28,8](	ON:= , 	OFF:= , 	LINK:=EL1008[28,8] , 	VALUE=> 	arRealAxisAdmin[42].i.HomeCali	);	(*	皮带2原点	*)
DI_[32,1](	ON:= , 	OFF:= , 	LINK:=EL1008[32,1] , 	VALUE=> 	arRealAxisAdmin[43].i.HomeCali	);	(*	皮带3原点	*)
DI_[32,2](	ON:= , 	OFF:= , 	LINK:=EL1008[32,2] , 	VALUE=> 	arDropBufferCyclinder[2].i.InSensor	);	(*	备用	*)
DI_[32,3](	ON:= , 	OFF:= , 	LINK:=EL1008[32,3] , 	VALUE=> 		);	(*	备用	*)
DI_[32,4](	ON:= , 	OFF:= , 	LINK:=EL1008[32,4] , 	VALUE=> 		);	(*	备用	*)
DI_[32,5](	ON:= , 	OFF:= , 	LINK:=EL1008[32,5] , 	VALUE=> 		);	(*	备用	*)
DI_[32,6](	ON:= , 	OFF:= , 	LINK:=EL1008[32,6] , 	VALUE=> 		);	(*	备用	*)
DI_[32,7](	ON:= , 	OFF:= , 	LINK:=EL1008[32,7] , 	VALUE=> 		);	(*	备用	*)
DI_[32,8](	ON:= , 	OFF:= , 	LINK:=EL1008[32,8] , 	VALUE=> 		);	(*	备用	*)

(*****************************************************************************************************)									
DO_[22,1](	ON:= , 	OFF:= , 	LINK=>EL2008[22,1] , 	VALUE:= 	arDropCylinder[31].o.ValveIn	);	(*	料仓31气缸原位	*)
DO_[22,2](	ON:= , 	OFF:= , 	LINK=>EL2008[22,2] , 	VALUE:= 	arDropCylinder[31].o.ValveOut	);	(*	料仓31气缸工作位	*)
DO_[22,3](	ON:= , 	OFF:= , 	LINK=>EL2008[22,3] , 	VALUE:= 	arDropCylinder[32].o.ValveIn	);	(*	料仓32气缸原位	*)
DO_[22,4](	ON:= , 	OFF:= , 	LINK=>EL2008[22,4] , 	VALUE:= 	arDropCylinder[32].o.ValveOut	);	(*	料仓32气缸工作位	*)
DO_[22,5](	ON:= , 	OFF:= , 	LINK=>EL2008[22,5] , 	VALUE:= 	arDropCylinder[33].o.ValveIn	);	(*	料仓33气缸原位	*)
DO_[22,6](	ON:= , 	OFF:= , 	LINK=>EL2008[22,6] , 	VALUE:= 	arDropCylinder[33].o.ValveOut	);	(*	料仓33气缸工作位	*)
DO_[22,7](	ON:= , 	OFF:= , 	LINK=>EL2008[22,7] , 	VALUE:= 	arDropCylinder[34].o.ValveIn	);	(*	料仓34气缸原位	*)
DO_[22,8](	ON:= , 	OFF:= , 	LINK=>EL2008[22,8] , 	VALUE:= 	arDropCylinder[34].o.ValveOut	);	(*	料仓34气缸工作位	*)
DO_[23,1](	ON:= , 	OFF:= , 	LINK=>EL2008[23,1] , 	VALUE:= 	arDropCylinder[35].o.ValveIn	);	(*	料仓35气缸原位	*)
DO_[23,2](	ON:= , 	OFF:= , 	LINK=>EL2008[23,2] , 	VALUE:= 	arDropCylinder[35].o.ValveOut	);	(*	料仓35气缸工作位	*)
DO_[23,3](	ON:= , 	OFF:= , 	LINK=>EL2008[23,3] , 	VALUE:= 	arDropCylinder[36].o.ValveIn	);	(*	料仓36气缸原位	*)
DO_[23,4](	ON:= , 	OFF:= , 	LINK=>EL2008[23,4] , 	VALUE:= 	arDropCylinder[36].o.ValveOut	);	(*	料仓36气缸工作位	*)
DO_[23,5](	ON:= , 	OFF:= , 	LINK=>EL2008[23,5] , 	VALUE:= 	arDropCylinder[37].o.ValveIn	);	(*	料仓37气缸原位	*)
DO_[23,6](	ON:= , 	OFF:= , 	LINK=>EL2008[23,6] , 	VALUE:= 	arDropCylinder[37].o.ValveOut	);	(*	料仓37气缸工作位	*)
DO_[23,7](	ON:= , 	OFF:= , 	LINK=>EL2008[23,7] , 	VALUE:= 	arDropCylinder[38].o.ValveIn	);	(*	料仓38气缸原位	*)
DO_[23,8](	ON:= , 	OFF:= , 	LINK=>EL2008[23,8] , 	VALUE:= 	arDropCylinder[38].o.ValveOut	);	(*	料仓38气缸工作位	*)
DO_[24,1](	ON:= , 	OFF:= , 	LINK=>EL2008[24,1] , 	VALUE:= 	arDropCylinder[39].o.ValveIn	);	(*	料仓39气缸原位	*)
DO_[24,2](	ON:= , 	OFF:= , 	LINK=>EL2008[24,2] , 	VALUE:= 	arDropCylinder[39].o.ValveOut	);	(*	料仓39气缸工作位	*)
DO_[24,3](	ON:= , 	OFF:= , 	LINK=>EL2008[24,3] , 	VALUE:= 	arDropCylinder[40].o.ValveIn	);	(*	料仓40气缸原位	*)
DO_[24,4](	ON:= , 	OFF:= , 	LINK=>EL2008[24,4] , 	VALUE:= 	arDropCylinder[40].o.ValveOut	);	(*	料仓40气缸工作位	*)
DO_[24,5](	ON:= , 	OFF:= , 	LINK=>EL2008[24,5] , 	VALUE:= 	arCounters[31].LineVibrator_Wrk	);	(*	料仓31直震启动	*)
DO_[24,6](	ON:= , 	OFF:= , 	LINK=>EL2008[24,6] , 	VALUE:= 	arCounters[31].CircleVibrator_Wrk	);	(*	料仓31圆震启动	*)
DO_[24,7](	ON:= , 	OFF:= , 	LINK=>EL2008[24,7] , 	VALUE:= 	arCounters[31].DropVibrator_Wrk	);	(*	料仓31落料启动	*)
DO_[24,8](	ON:= , 	OFF:= , 	LINK=>EL2008[24,8] , 	VALUE:= 	arCounters[32].LineVibrator_Wrk	);	(*	料仓32直震启动	*)
DO_[25,1](	ON:= , 	OFF:= , 	LINK=>EL2008[25,1] , 	VALUE:= 	arCounters[32].CircleVibrator_Wrk	);	(*	料仓32圆震启动	*)
DO_[25,2](	ON:= , 	OFF:= , 	LINK=>EL2008[25,2] , 	VALUE:= 	arCounters[32].DropVibrator_Wrk	);	(*	料仓32落料启动	*)
DO_[25,3](	ON:= , 	OFF:= , 	LINK=>EL2008[25,3] , 	VALUE:= 	arCounters[33].LineVibrator_Wrk	);	(*	料仓33直震启动	*)
DO_[25,4](	ON:= , 	OFF:= , 	LINK=>EL2008[25,4] , 	VALUE:= 	arCounters[33].CircleVibrator_Wrk	);	(*	料仓33圆震启动	*)
DO_[25,5](	ON:= , 	OFF:= , 	LINK=>EL2008[25,5] , 	VALUE:= 	arCounters[33].DropVibrator_Wrk	);	(*	料仓33落料启动	*)
DO_[25,6](	ON:= , 	OFF:= , 	LINK=>EL2008[25,6] , 	VALUE:= 	arCounters[34].LineVibrator_Wrk	);	(*	料仓34直震启动	*)
DO_[25,7](	ON:= , 	OFF:= , 	LINK=>EL2008[25,7] , 	VALUE:= 	arCounters[34].CircleVibrator_Wrk	);	(*	料仓34圆震启动	*)
DO_[25,8](	ON:= , 	OFF:= , 	LINK=>EL2008[25,8] , 	VALUE:= 	arCounters[34].DropVibrator_Wrk	);	(*	料仓34落料启动	*)
DO_[26,1](	ON:= , 	OFF:= , 	LINK=>EL2008[26,1] , 	VALUE:= 	arCounters[35].LineVibrator_Wrk	);	(*	料仓35直震启动	*)
DO_[26,2](	ON:= , 	OFF:= , 	LINK=>EL2008[26,2] , 	VALUE:= 	arCounters[35].CircleVibrator_Wrk	);	(*	料仓35圆震启动	*)
DO_[26,3](	ON:= , 	OFF:= , 	LINK=>EL2008[26,3] , 	VALUE:= 	arCounters[35].DropVibrator_Wrk	);	(*	料仓35落料启动	*)
DO_[26,4](	ON:= , 	OFF:= , 	LINK=>EL2008[26,4] , 	VALUE:= 	arCounters[36].LineVibrator_Wrk	);	(*	料仓36直震启动	*)
DO_[26,5](	ON:= , 	OFF:= , 	LINK=>EL2008[26,5] , 	VALUE:= 	arCounters[36].CircleVibrator_Wrk	);	(*	料仓36圆震启动	*)
DO_[26,6](	ON:= , 	OFF:= , 	LINK=>EL2008[26,6] , 	VALUE:= 	arCounters[36].DropVibrator_Wrk	);	(*	料仓36落料启动	*)
DO_[26,7](	ON:= , 	OFF:= , 	LINK=>EL2008[26,7] , 	VALUE:= 	arCounters[37].LineVibrator_Wrk	);	(*	料仓37直震启动	*)
DO_[26,8](	ON:= , 	OFF:= , 	LINK=>EL2008[26,8] , 	VALUE:= 	arCounters[37].CircleVibrator_Wrk	);	(*	料仓37圆震启动	*)
DO_[27,1](	ON:= , 	OFF:= , 	LINK=>EL2008[27,1] , 	VALUE:= 	arCounters[37].DropVibrator_Wrk	);	(*	料仓37落料启动	*)
DO_[27,2](	ON:= , 	OFF:= , 	LINK=>EL2008[27,2] , 	VALUE:= 	arCounters[38].LineVibrator_Wrk	);	(*	料仓38直震启动	*)
DO_[27,3](	ON:= , 	OFF:= , 	LINK=>EL2008[27,3] , 	VALUE:= 	arCounters[38].CircleVibrator_Wrk	);	(*	料仓38圆震启动	*)
DO_[27,4](	ON:= , 	OFF:= , 	LINK=>EL2008[27,4] , 	VALUE:= 	arCounters[38].DropVibrator_Wrk	);	(*	料仓38落料启动	*)
DO_[27,5](	ON:= , 	OFF:= , 	LINK=>EL2008[27,5] , 	VALUE:= 	arCounters[39].LineVibrator_Wrk	);	(*	料仓39直震启动	*)
DO_[27,6](	ON:= , 	OFF:= , 	LINK=>EL2008[27,6] , 	VALUE:= 	arCounters[39].CircleVibrator_Wrk	);	(*	料仓39圆震启动	*)
DO_[27,7](	ON:= , 	OFF:= , 	LINK=>EL2008[27,7] , 	VALUE:= 	arCounters[39].DropVibrator_Wrk	);	(*	料仓39落料启动	*)
DO_[27,8](	ON:= , 	OFF:= , 	LINK=>EL2008[27,8] , 	VALUE:= 	arCounters[40].LineVibrator_Wrk	);	(*	料仓40直震启动	*)
DO_[28,1](	ON:= , 	OFF:= , 	LINK=>EL2008[28,1] , 	VALUE:= 	arCounters[40].CircleVibrator_Wrk	);	(*	料仓40圆震启动	*)
DO_[28,2](	ON:= , 	OFF:= , 	LINK=>EL2008[28,2] , 	VALUE:= 	arCounters[40].DropVibrator_Wrk	);	(*	料仓40落料启动	*)
DO_[28,3](	ON:= , 	OFF:= , 	LINK=>EL2008[28,3] , 	VALUE:= 	glb_arLightRelay_UN01[2]	);	(*	数粒系统2设备照明继电器	*)
DO_[28,4](	ON:= , 	OFF:= , 	LINK=>EL2008[28,4] , 	VALUE:= 		);	(*	备用	*)
DO_[28,5](	ON:= , 	OFF:= , 	LINK=>EL2008[28,5] , 	VALUE:= 		);	(*	备用	*)
DO_[28,6](	ON:= , 	OFF:= , 	LINK=>EL2008[28,6] , 	VALUE:= 		);	(*	备用	*)
DO_[28,7](	ON:= , 	OFF:= , 	LINK=>EL2008[28,7] , 	VALUE:= 		);	(*	备用	*)
DO_[28,8](	ON:= , 	OFF:= , 	LINK=>EL2008[28,8] , 	VALUE:= 		);	(*	备用	*)
									
{endregion}
END_ACTION

ACTION CP07:
{region CP07}
DI_[33,1]	(	ON:= , 	OFF:= , 	LINK:=EL1008[33,1] , 	VALUE=> glb_bModeSwitch_UN01		);	(*	手自动选择	*)
DI_[33,2]	(	ON:= , 	OFF:= , 	LINK:=EL1008[33,2] , 	VALUE=> glb_bStartButton_UN01		);	(*	启动	*)
DI_[33,3]	(	ON:= , 	OFF:= , 	LINK:=EL1008[33,3] , 	VALUE=> glb_bStopButton_UN01		);	(*	停止	*)
DI_[33,4]	(	ON:= , 	OFF:= , 	LINK:=EL1008[33,4] , 	VALUE=> glb_bResetButton_UN01		);	(*	复位	*)
DI_[33,5]	(	ON:= , 	OFF:= , 	LINK:=EL1008[33,5] , 	VALUE=> glb_diEstopButton_UN01.0		);	(*	急停	*)
DI_[33,6]	(	ON:= , 	OFF:= , 	LINK:=EL1008[33,6] , 	VALUE=> glb_bAirFeedback_UN01[1]		);	(*	总气压反馈	*)
DI_[33,7]	(	ON:= , 	OFF:= , 	LINK:=EL1008[33,7] , 	VALUE=> arSafeDoorSts[19]		);	(*	安全门19	*)
DI_[33,8]	(	ON:= , 	OFF:= , 	LINK:=EL1008[33,8] , 	VALUE=> arSafeDoorSts[20]		);	(*	安全门20	*)
DI_[34,1]	(	ON:= , 	OFF:= , 	LINK:=EL1008[34,1] , 	VALUE=> arSafeDoorSts[21]		);	(*	安全门21	*)
DI_[34,2]	(	ON:= , 	OFF:= , 	LINK:=EL1008[34,2] , 	VALUE=> arSafeDoorSts[22]		);	(*	安全门22	*)
DI_[34,3]	(	ON:= , 	OFF:= , 	LINK:=EL1008[34,3] , 	VALUE=> arSafeDoorSts[23]		);	(*	安全门23	*)
DI_[34,4]	(	ON:= , 	OFF:= , 	LINK:=EL1008[34,4] , 	VALUE=> arPackCylinder[41].i.InSensor		    );	(*	铝杯检测气缸In	*)
DI_[34,5]	(	ON:= , 	OFF:= , 	LINK:=EL1008[34,5] , 	VALUE=> arPackCylinder[41].i.OutSensor		    );	(*	铝杯检测气缸OUT	*)
DI_[34,6]	(	ON:= , 	OFF:= , 	LINK:=EL1008[34,6] , 	VALUE=> arPackSensor[41].i.Link	    	    );	(*铝杯检测接近开关1		*)
DI_[34,7]	(	ON:= , 	OFF:= , 	LINK:=EL1008[34,7] , 	VALUE=> arPackSensor[42].i.Link			    );	(*铝杯检测接近开关2		*)
DI_[34,8]	(	ON:= , 	OFF:= , 	LINK:=EL1008[34,8] , 	VALUE=> arPackSensor[43].i.Link			    );	(*铝杯检测接近开关3		*)
DI_[35,1]	(	ON:= , 	OFF:= , 	LINK:=EL1008[35,1] , 	VALUE=> arPackSensor[44].i.Link	        	);	(*铝杯检测接近开关4	    *)
DI_[35,2]	(	ON:= , 	OFF:= , 	LINK:=EL1008[35,2] , 	VALUE=> arPackSensor[45].i.Link	    		);	(*铝杯检测接近开关5  	*)
DI_[35,3]	(	ON:= , 	OFF:= , 	LINK:=EL1008[35,3] , 	VALUE=> arPackSensor[46].i.Link	    		);	(*铝杯检测接近开关6 	*)
DI_[35,4]	(	ON:= , 	OFF:= , 	LINK:=EL1008[35,4] , 	VALUE=> arPackSensor[47].i.Link	    		);	(*铝杯检测接近开关7  	*)
DI_[35,5]	(	ON:= , 	OFF:= , 	LINK:=EL1008[35,5] , 	VALUE=>     		);	(*	*)
DI_[35,6]	(	ON:= , 	OFF:= , 	LINK:=EL1008[35,6] , 	VALUE=>     		);	(*	*)
DI_[35,7]	(	ON:= , 	OFF:= , 	LINK:=EL1008[35,7] , 	VALUE=>     		);	(*	*)
DI_[35,8]	(	ON:= , 	OFF:= , 	LINK:=EL1008[35,8] , 	VALUE=> 		    );	(*	*)
DI_[36,1]	(	ON:= , 	OFF:= , 	LINK:=EL1008[36,1] , 	VALUE=> arPackVacuum[1].i.Sensor		);	(*	拉料气缸1真空反馈	*)
DI_[36,2]	(	ON:= , 	OFF:= , 	LINK:=EL1008[36,2] , 	VALUE=> arPackVacuum[2].i.Sensor		);	(*	拉料气缸2真空反馈	*)
DI_[36,3]	(	ON:= , 	OFF:= , 	LINK:=EL1008[36,3] , 	VALUE=> arPackVacuum[3].i.Sensor		);	(*	拉料气缸3真空反馈	*)
DI_[36,4]	(	ON:= , 	OFF:= , 	LINK:=EL1008[36,4] , 	VALUE=> arPackVacuum[4].i.Sensor		);	(*	拉料气缸4真空反馈	*)
DI_[36,5]	(	ON:= , 	OFF:= , 	LINK:=EL1008[36,5] , 	VALUE=> arPackVacuum[5].i.Sensor		);	(*	拉料气缸5真空反馈	*)
DI_[36,6]	(	ON:= , 	OFF:= , 	LINK:=EL1008[36,6] , 	VALUE=> arPackVacuum[6].i.Sensor		);	(*	拉料气缸6真空反馈	*)
DI_[36,7]	(	ON:= , 	OFF:= , 	LINK:=EL1008[36,7] , 	VALUE=> arPackVacuum[7].i.Sensor		);	(*	拉料气缸7真空反馈	*)
DI_[36,8]	(	ON:= , 	OFF:= , 	LINK:=EL1008[36,8] , 	VALUE=> arPackVacuum[11].i.Sensor		);	(*	平移气缸1真空反馈	*)
DI_[37,1]	(	ON:= , 	OFF:= , 	LINK:=EL1008[37,1] , 	VALUE=> arPackVacuum[12].i.Sensor		);	(*	平移气缸2真空反馈	*)
DI_[37,2]	(	ON:= , 	OFF:= , 	LINK:=EL1008[37,2] , 	VALUE=> arPackVacuum[13].i.Sensor		);	(*	平移气缸3真空反馈	*)
DI_[37,3]	(	ON:= , 	OFF:= , 	LINK:=EL1008[37,3] , 	VALUE=> arPackVacuum[14].i.Sensor		);	(*	平移气缸4真空反馈	*)
DI_[37,4]	(	ON:= , 	OFF:= , 	LINK:=EL1008[37,4] , 	VALUE=> arPackVacuum[15].i.Sensor		);	(*	平移气缸5真空反馈	*)
DI_[37,5]	(	ON:= , 	OFF:= , 	LINK:=EL1008[37,5] , 	VALUE=> arPackVacuum[16].i.Sensor		);	(*	平移气缸6真空反馈	*)
DI_[37,6]	(	ON:= , 	OFF:= , 	LINK:=EL1008[37,6] , 	VALUE=> arPackVacuum[17].i.Sensor		);	(*	平移气缸7真空反馈	*)
DI_[37,7]	(	ON:= , 	OFF:= , 	LINK:=EL1008[37,7] , 	VALUE=> 		);	(*	*)
DI_[37,8]	(	ON:= , 	OFF:= , 	LINK:=EL1008[37,8] , 	VALUE=> 		);	(*	*)
	 
(*************************************************************************************************************)
DO_[29,1]	(	ON:= , 	OFF:= , 	LINK=>EL2008[29,1] , 	VALUE:= glb_arLightRed_UN01[3] 		);	(*	三色灯红	*)
DO_[29,2]	(	ON:= , 	OFF:= , 	LINK=>EL2008[29,2] , 	VALUE:= glb_arLightYellow_UN01[3] 		);	(*	三色灯黄	*)
DO_[29,3]	(	ON:= , 	OFF:= , 	LINK=>EL2008[29,3] , 	VALUE:= glb_arLightGreen_UN01[3]		);	(*	三色灯绿	*)
DO_[29,4]	(	ON:= , 	OFF:= , 	LINK=>EL2008[29,4] , 	VALUE:= glb_arLightAlarm_UN01[3]		);	(*	三色灯蜂鸣器	*)
DO_[29,5]	(	ON:= , 	OFF:= , 	LINK=>EL2008[29,5] , 	VALUE:= glb_bPackAirValve_UN01 		);	(*	总气压阀	*)
DO_[29,6]	(	ON:= , 	OFF:= , 	LINK=>EL2008[29,6] , 	VALUE:= arPackMotor[1].Forward		);	(*	力矩电机正转	*)
DO_[29,7]	(	ON:= , 	OFF:= , 	LINK=>EL2008[29,7] , 	VALUE:= arPackMotor[1].Backward		);	(*	力矩电机反转	*)
DO_[29,8]	(	ON:= , 	OFF:= , 	LINK=>EL2008[29,8] , 	VALUE:= arPackHeatRealy[1]		);	(*	加热棒1	*)
DO_[30,1]	(	ON:= , 	OFF:= , 	LINK=>EL2008[30,1] , 	VALUE:= arPackHeatRealy[2]		);	(*	加热棒2	*)
DO_[30,2]	(	ON:= , 	OFF:= , 	LINK=>EL2008[30,2] , 	VALUE:= arPackHeatRealy[3]		);	(*	加热棒3	*)
DO_[30,3]	(	ON:= , 	OFF:= , 	LINK=>EL2008[30,3] , 	VALUE:= arPackHeatRealy[4]		);	(*	加热棒4	*)
DO_[30,4]	(	ON:= , 	OFF:= , 	LINK=>EL2008[30,4] , 	VALUE:= arPackHeatRealy[5]		);	(*	加热棒5	*)
DO_[30,5]	(	ON:= , 	OFF:= , 	LINK=>EL2008[30,5] , 	VALUE:= arPackHeatRealy[6]		);	(*	加热棒6	*)
DO_[30,6]	(	ON:= , 	OFF:= , 	LINK=>EL2008[30,6] , 	VALUE:= arPackHeatRealy[7]		);	(*	加热棒7	*)
DO_[30,7]	(	ON:= , 	OFF:= , 	LINK=>EL2008[30,7] , 	VALUE:= arPackVacuum[1].o.ValveIn		);	(*	拉料气缸1真空吸	*)
DO_[30,8]	(	ON:= , 	OFF:= , 	LINK=>EL2008[30,8] , 	VALUE:= arPackVacuum[1].o.ValveOut		);	(*	拉料气缸1真空吹	*)
DO_[31,1]	(	ON:= , 	OFF:= , 	LINK=>EL2008[31,1] , 	VALUE:= arPackVacuum[11].o.ValveIn	);	(*	平移真空1吸	*)
DO_[31,2]	(	ON:= , 	OFF:= , 	LINK=>EL2008[31,2] , 	VALUE:= arPackVacuum[11].o.ValveOut		);	(*	平移真空1吹	*)
DO_[31,3]	(	ON:= , 	OFF:= , 	LINK=>EL2008[31,3] , 	VALUE:= glb_bStartBottonLight_UN01		);	(*	启动按钮指示灯	*)
DO_[31,4]	(	ON:= , 	OFF:= , 	LINK=>EL2008[31,4] , 	VALUE:= glb_bStopBottonLight_UN01			);	(*	停止按钮指示灯	*)
DO_[31,5]	(	ON:= , 	OFF:= , 	LINK=>EL2008[31,5] , 	VALUE:= glb_bResetBottonLight_UN01		);	(*	复位按钮指示灯	*)
DO_[31,6]	(	ON:= , 	OFF:= , 	LINK=>EL2008[31,6] , 	VALUE:= arPackCylinder[17].o.ValveOut		);	(*	药盒封口气缸OUT	*)
DO_[31,7]	(	ON:= , 	OFF:= , 	LINK=>EL2008[31,7] , 	VALUE:= arPackHeatRealy[8]		);	(*	加热棒8	*)
DO_[31,8]	(	ON:= , 	OFF:= , 	LINK=>EL2008[31,8] , 	VALUE:= arPackCylinder[18].o.ValveOut		);	(*	药盒封口2上气缸OUT	*)
DO_[32,1]	(	ON:= , 	OFF:= , 	LINK=>EL2008[32,1] , 	VALUE:= arPackCylinder[19].o.ValveOut		);	(*	药盒封口2下气缸OUT	*)
DO_[32,2]	(	ON:= , 	OFF:= , 	LINK=>EL2008[32,2] , 	VALUE:= arPackCylinder[20].o.ValveOut		);	(*	剔除气缸20210420	*)
DO_[32,3]	(	ON:= , 	OFF:= , 	LINK=>EL2008[32,3] , 	VALUE:= 		);	(*	预留	*)
DO_[32,4]	(	ON:= , 	OFF:= , 	LINK=>EL2008[32,4] , 	VALUE:= 		);	(*	预留	*)
DO_[32,5]	(	ON:= , 	OFF:= , 	LINK=>EL2008[32,5] , 	VALUE:= 		);	(*	预留	*)
DO_[32,6]	(	ON:= , 	OFF:= , 	LINK=>EL2008[32,6] , 	VALUE:= 		);	(*	预留	*)
DO_[32,7]	(	ON:= , 	OFF:= , 	LINK=>EL2008[32,7] , 	VALUE:= 		);	(*	预留	*)
DO_[32,8]	(	ON:= , 	OFF:= , 	LINK=>EL2008[32,8] , 	VALUE:= 		);	(*	预留	*)
	 					
{endregion}
END_ACTION

ACTION CPX1:
{region 现场IO1}
DI_[50,1](	ON:= , 	OFF:= , 	LINK:=CPX8_1[1,1] , 	VALUE=> arPackCylinder[17].i.InSensor		);	(*	冲裁气缸	IN	*)
DI_[50,2](	ON:= , 	OFF:= , 	LINK:=CPX8_1[1,2] , 	VALUE=> arPackCylinder[17].i.OutSensor		);	(*	冲裁气缸	OUT	*)
DI_[50,3](	ON:= , 	OFF:= , 	LINK:=CPX8_1[1,3] , 	VALUE=> arPackCylinder[15].i.InSensor		);	(*	料板支撑气缸	IN	*)
DI_[50,4](	ON:= , 	OFF:= , 	LINK:=CPX8_1[1,4] , 	VALUE=> arPackCylinder[15].i.OutSensor		);	(*	料板支撑气缸	OUT	*)
DI_[50,5](	ON:= , 	OFF:= , 	LINK:=CPX8_1[1,5] , 	VALUE=> arPackCylinder[14].i.InSensor		);	(*	移载无杆气缸	IN	*)
DI_[50,6](	ON:= , 	OFF:= , 	LINK:=CPX8_1[1,6] , 	VALUE=> arPackCylinder[14].i.OutSensor		);	(*	移载无杆气缸	OUT	*)
DI_[50,7](	ON:= , 	OFF:= , 	LINK:=CPX8_1[1,7] , 	VALUE=> arPackCylinder[16].i.InSensor		);	(*	移载垂移滑台	IN	*)
DI_[50,8](	ON:= , 	OFF:= , 	LINK:=CPX8_1[1,8] , 	VALUE=> arPackCylinder[16].i.OutSensor		);	(*	移载垂移滑台	OUT	*)
DI_[51,1](	ON:= , 	OFF:= , 	LINK:=CPX8_1[2,1] , 	VALUE=> arPackCylinder[13].i.InSensor		);	(*	单排旋转气缸	IN	*)
DI_[51,2](	ON:= , 	OFF:= , 	LINK:=CPX8_1[2,2] , 	VALUE=> arPackCylinder[13].i.OutSensor		);	(*	单排旋转气缸	OUT	*)
DI_[51,3](	ON:= , 	OFF:= , 	LINK:=CPX8_1[2,3] , 	VALUE=> arRealAxisAdmin[46].i.HomeCali	    );	(*	皮带6原点		*)
DI_[51,4](	ON:= , 	OFF:= , 	LINK:=CPX8_1[2,4] , 	VALUE=> arPackCylinder[10].i.InSensor		);	(*	封口上气缸 IN   *)arPackCylinder[10].i.OutSensor:=NOT arPackCylinder[10].i.InSensor;
DI_[51,5](	ON:= , 	OFF:= , 	LINK:=CPX8_1[2,5] , 	VALUE=> arPackCylinder[18].i.InSensor		);	(*	封口2上气缸 IN  *)arPackCylinder[18].i.OutSensor:=NOT arPackCylinder[18].i.InSensor;
DI_[51,6](	ON:= , 	OFF:= , 	LINK:=CPX8_1[2,6] , 	VALUE=> arPackCylinder[11].i.InSensor		);	(*	封口下气缸 IN 	*)
DI_[51,7](	ON:= , 	OFF:= , 	LINK:=CPX8_1[2,7] , 	VALUE=> arPackCylinder[11].i.OutSensor		);	(*	封口下气缸 OUT  *)
DI_[51,8](	ON:= , 	OFF:= , 	LINK:=CPX8_1[2,8] , 	VALUE=> arRealAxisAdmin[48].i.HomeCali     	);	(*	皮带7原点         20210420   	*)
DI_[52,1](	ON:= , 	OFF:= , 	LINK:=CPX8_1[3,1] , 	VALUE=> arPackCylinder[1].i.InSensor		);	(*	吸盒气缸1	IN	*)
DI_[52,2](	ON:= , 	OFF:= , 	LINK:=CPX8_1[3,2] , 	VALUE=> 		);	(*	吸盒气缸1	OUT arPackCylinder[1].i.OutSensor	*)
DI_[52,3](	ON:= , 	OFF:= , 	LINK:=CPX8_1[3,3] , 	VALUE=> arPackCylinder[2].i.InSensor		);	(*	吸盒气缸2	IN	*)
DI_[52,4](	ON:= , 	OFF:= , 	LINK:=CPX8_1[3,4] , 	VALUE=> 		);	(*	吸盒气缸2	OUT	arPackCylinder[2].i.OutSensor*)
DI_[52,5](	ON:= , 	OFF:= , 	LINK:=CPX8_1[3,5] , 	VALUE=> arPackCylinder[3].i.InSensor		);	(*	吸盒气缸3	IN	*)
DI_[52,6](	ON:= , 	OFF:= , 	LINK:=CPX8_1[3,6] , 	VALUE=> 		);	(*	吸盒气缸3	OUT	arPackCylinder[3].i.OutSensor*)
DI_[52,7](	ON:= , 	OFF:= , 	LINK:=CPX8_1[3,7] , 	VALUE=> arPackCylinder[4].i.InSensor		);	(*	吸盒气缸4	IN	*)
DI_[52,8](	ON:= , 	OFF:= , 	LINK:=CPX8_1[3,8] , 	VALUE=> 		);	(*	吸盒气缸4	OUT	arPackCylinder[4].i.OutSensor*)
DI_[53,1](	ON:= , 	OFF:= , 	LINK:=CPX8_1[4,1] , 	VALUE=> arPackCylinder[5].i.InSensor		);	(*	吸盒气缸5	IN	*)
DI_[53,2](	ON:= , 	OFF:= , 	LINK:=CPX8_1[4,2] , 	VALUE=> 		);	(*	吸盒气缸5	OUT	arPackCylinder[5].i.OutSensor*)
DI_[53,3](	ON:= , 	OFF:= , 	LINK:=CPX8_1[4,3] , 	VALUE=> arPackCylinder[6].i.InSensor		);	(*	吸盒气缸6	IN	*)
DI_[53,4](	ON:= , 	OFF:= , 	LINK:=CPX8_1[4,4] , 	VALUE=> 		);	(*	吸盒气缸6	OUT	arPackCylinder[6].i.OutSensor*)
DI_[53,5](	ON:= , 	OFF:= , 	LINK:=CPX8_1[4,5] , 	VALUE=> arPackCylinder[7].i.InSensor	    );	(*	吸盒气缸7	IN	*)
DI_[53,6](	ON:= , 	OFF:= , 	LINK:=CPX8_1[4,6] , 	VALUE=> 		);	(*	吸盒气缸7	OUT	arPackCylinder[7].i.OutSensor*)
DI_[53,7](	ON:= , 	OFF:= , 	LINK:=CPX8_1[4,7] , 	VALUE=> arPackCylinder[19].i.InSensor		);	(*	封口2下气缸 IN	*)
DI_[53,8](	ON:= , 	OFF:= , 	LINK:=CPX8_1[4,8] , 	VALUE=> arPackCylinder[19].i.OutSensor		);	(*	封口2下气缸 OUT	*)//热封2
DI_[54,1](	ON:= , 	OFF:= , 	LINK:=CPX8_1[5,1] , 	VALUE=> arPackCylinder[8].i.InSensor		);	(*	放药气缸	IN	*)
DI_[54,2](	ON:= , 	OFF:= , 	LINK:=CPX8_1[5,2] , 	VALUE=> arPackCylinder[8].i.OutSensor		);	(*	放药气缸	OUT	*)
DI_[54,3](	ON:= , 	OFF:= , 	LINK:=CPX8_1[5,3] , 	VALUE=> arPackCylinder[12].i.InSensor		);	(*	药品输送气缸		*)
DI_[54,4](	ON:= , 	OFF:= , 	LINK:=CPX8_1[5,4] , 	VALUE=> 		);	(*	药品输送气缸	OUT	*)
DI_[54,5](	ON:= , 	OFF:= , 	LINK:=CPX8_1[5,5] , 	VALUE=> arPackCylinder[9].i.InSensor		);	(*	工位转换气缸	IN	*)
DI_[54,6](	ON:= , 	OFF:= , 	LINK:=CPX8_1[5,6] , 	VALUE=> arPackCylinder[9].i.OutSensor		);	(*	工位转换气缸	OUT	*)
DI_[54,7](	ON:= , 	OFF:= , 	LINK:=CPX8_1[5,7] , 	VALUE=> 		);	(*			*)
DI_[54,8](	ON:= , 	OFF:= , 	LINK:=CPX8_1[5,8] , 	VALUE=> 		);	(*			*)
DI_[55,1](	ON:= , 	OFF:= , 	LINK:=CPX8_1[6,1] , 	VALUE=> arPackSensor[1].i.Link		);	(*	盒子检测光电1		*)
DI_[55,2](	ON:= , 	OFF:= , 	LINK:=CPX8_1[6,2] , 	VALUE=> arPackSensor[2].i.Link		);	(*	盒子检测光电2		*)
DI_[55,3](	ON:= , 	OFF:= , 	LINK:=CPX8_1[6,3] , 	VALUE=> arPackSensor[3].i.Link		);	(*	盒子检测光电3		*)
DI_[55,4](	ON:= , 	OFF:= , 	LINK:=CPX8_1[6,4] , 	VALUE=> arPackSensor[4].i.Link		);	(*	盒子检测光电4		*)
DI_[55,5](	ON:= , 	OFF:= , 	LINK:=CPX8_1[6,5] , 	VALUE=> arPackSensor[5].i.Link		);	(*	盒子检测光电5		*)
DI_[55,6](	ON:= , 	OFF:= , 	LINK:=CPX8_1[6,6] , 	VALUE=> arPackSensor[6].i.Link		);	(*	盒子检测光电6		*)
DI_[55,7](	ON:= , 	OFF:= , 	LINK:=CPX8_1[6,7] , 	VALUE=> arPackSensor[7].i.Link		);	(*	盒子检测光电7		*)
DI_[55,8](	ON:= , 	OFF:= , 	LINK:=CPX8_1[6,8] , 	VALUE=> arPackSensor[8].i.Link		);	(*	盒子检测光电8		*)
DI_[56,1](	ON:= , 	OFF:= , 	LINK:=CPX8_1[7,1] , 	VALUE=> arPackSensor[9].i.Link		);	(*	盒子检测光电9		*)
DI_[56,2](	ON:= , 	OFF:= , 	LINK:=CPX8_1[7,2] , 	VALUE=> arPackSensor[10].i.Link		);	(*	盒子检测光电10		*)
DI_[56,3](	ON:= , 	OFF:= , 	LINK:=CPX8_1[7,3] , 	VALUE=> arPackSensor[11].i.Link		);	(*	盒子检测光电11		*)
DI_[56,4](	ON:= , 	OFF:= , 	LINK:=CPX8_1[7,4] , 	VALUE=> arPackSensor[12].i.Link		);	(*	盒子检测光电12		*)
DI_[56,5](	ON:= , 	OFF:= , 	LINK:=CPX8_1[7,5] , 	VALUE=> arPackSensor[13].i.Link		);	(*	盒子检测光电13		*)
DI_[56,6](	ON:= , 	OFF:= , 	LINK:=CPX8_1[7,6] , 	VALUE=> arPackSensor[14].i.Link		);	(*	盒子检测光电14		*)
DI_[56,7](	ON:= , 	OFF:= , 	LINK:=CPX8_1[7,7] , 	VALUE=> arRealAxisAdmin[44].i.HomeCali		);	(*	差速线接近开关1		*)
DI_[56,8](	ON:= , 	OFF:= , 	LINK:=CPX8_1[7,8] , 	VALUE=> arRealAxisAdmin[45].i.HomeCali		);	(*	差速线接近开关2		*)

{endregion}
END_ACTION

ACTION WPI1:
{region WPI_1}
DO_[50,1]	(	ON:= , 	OFF:= , 	LINK=>WPI_1[1,1] , 	VALUE:= arPackCylinder[1].o.ValveIn	);	//	吸盒气缸1In
DO_[50,2]	(	ON:= , 	OFF:= , 	LINK=>WPI_1[1,2] , 	VALUE:= arPackCylinder[1].o.ValveOut	);	//	吸盒气缸1Out
DO_[50,3]	(	ON:= , 	OFF:= , 	LINK=>WPI_1[1,3] , 	VALUE:= arPackCylinder[2].o.ValveIn	);	//	吸盒气缸2In
DO_[50,4]	(	ON:= , 	OFF:= , 	LINK=>WPI_1[1,4] , 	VALUE:= arPackCylinder[2].o.ValveOut	);	//	吸盒气缸2Out
DO_[50,5]	(	ON:= , 	OFF:= , 	LINK=>WPI_1[1,5] , 	VALUE:= arPackCylinder[3].o.ValveIn	);	//	吸盒气缸3In
DO_[50,6]	(	ON:= , 	OFF:= , 	LINK=>WPI_1[1,6] , 	VALUE:= arPackCylinder[3].o.ValveOut	);	//	吸盒气缸3Out
DO_[50,7]	(	ON:= , 	OFF:= , 	LINK=>WPI_1[1,7] , 	VALUE:= arPackCylinder[4].o.ValveIn	);	//	吸盒气缸4In
DO_[50,8]	(	ON:= , 	OFF:= , 	LINK=>WPI_1[1,8] , 	VALUE:= arPackCylinder[4].o.ValveOut	);	//	吸盒气缸4Out
DO_[51,1]	(	ON:= , 	OFF:= , 	LINK=>WPI_1[2,1] , 	VALUE:= arPackCylinder[5].o.ValveIn	);	//	吸盒气缸5In
DO_[51,2]	(	ON:= , 	OFF:= , 	LINK=>WPI_1[2,2] , 	VALUE:= arPackCylinder[5].o.ValveOut	);	//	吸盒气缸5Out
DO_[51,3]	(	ON:= , 	OFF:= , 	LINK=>WPI_1[2,3] , 	VALUE:= arPackCylinder[6].o.ValveIn	);	//	吸盒气缸6In
DO_[51,4]	(	ON:= , 	OFF:= , 	LINK=>WPI_1[2,4] , 	VALUE:= arPackCylinder[6].o.ValveOut	);	//	吸盒气缸6Out
DO_[51,5]	(	ON:= , 	OFF:= , 	LINK=>WPI_1[2,5] , 	VALUE:= arPackCylinder[7].o.ValveIn	    );	//	吸盒气缸7In
DO_[51,6]	(	ON:= , 	OFF:= , 	LINK=>WPI_1[2,6] , 	VALUE:= arPackCylinder[7].o.ValveOut	);	//	吸盒气缸7Out
DO_[51,7]	(	ON:= , 	OFF:= , 	LINK=>WPI_1[2,7] , 	VALUE:= arPackCylinder[8].o.ValveIn   	);	//	放药气缸In
DO_[51,8]	(	ON:= , 	OFF:= , 	LINK=>WPI_1[2,8] , 	VALUE:= arPackCylinder[8].o.ValveOut	);	//	放药气缸Out
DO_[52,1]	(	ON:= , 	OFF:= , 	LINK=>WPI_1[3,1] ,	VALUE:= arPackCylinder[9].o.ValveIn	    );	//	工位转换In
DO_[52,2]	(	ON:= , 	OFF:= , 	LINK=>WPI_1[3,2] ,	VALUE:= arPackCylinder[9].o.ValveOut	);	//	工位转换Out
DO_[52,3]	(	ON:= , 	OFF:= , 	LINK=>WPI_1[3,3] ,	VALUE:= arPackCylinder[10].o.ValveIn	);	//	封口上气缸IN
DO_[52,4]	(	ON:= , 	OFF:= , 	LINK=>WPI_1[3,4] ,	VALUE:= arPackCylinder[10].o.ValveOut	);	//	封口上气缸Out
DO_[52,5]	(	ON:= , 	OFF:= , 	LINK=>WPI_1[3,5] ,	VALUE:= arPackCylinder[11].o.ValveIn	);	//	封口下气缸IN
DO_[52,6]	(	ON:= , 	OFF:= , 	LINK=>WPI_1[3,6] ,	VALUE:= arPackCylinder[11].o.ValveOut	);	//	封口下气缸OUT
DO_[52,7]	(	ON:= , 	OFF:= , 	LINK=>WPI_1[3,7] ,	VALUE:= arPackCylinder[12].o.ValveIn	);	//	药品输送In
DO_[52,8]	(	ON:= , 	OFF:= , 	LINK=>WPI_1[3,8] ,	VALUE:= arPackCylinder[12].o.ValveOut	);	//	药品输送Out
DO_[53,1]	(	ON:= , 	OFF:= , 	LINK=>WPI_1[4,1] ,	VALUE:= 	);		
DO_[53,2]	(	ON:= , 	OFF:= , 	LINK=>WPI_1[4,2] ,	VALUE:= 	);		
DO_[53,3]	(	ON:= , 	OFF:= , 	LINK=>WPI_1[4,3] ,	VALUE:= 	);		
DO_[53,4]	(	ON:= , 	OFF:= , 	LINK=>WPI_1[4,4] ,	VALUE:= 	);		
DO_[53,5]	(	ON:= , 	OFF:= , 	LINK=>WPI_1[4,5] ,	VALUE:= 	);		
DO_[53,6]	(	ON:= , 	OFF:= , 	LINK=>WPI_1[4,6] ,	VALUE:= 	);		
DO_[53,7]	(	ON:= , 	OFF:= , 	LINK=>WPI_1[4,7] ,	VALUE:= 	);		
DO_[53,8]	(	ON:= , 	OFF:= , 	LINK=>WPI_1[4,8] ,	VALUE:= 	);		
{endregion}
END_ACTION

ACTION WPI2:
{region WPI_2}
DO_[54,1] 	 (	ON:= , 	OFF:= , 	LINK=>WPI_2[1,1] ,	VALUE:= arPackCylinder[16].o.ValveOut		);	(* 单控阀	单排旋转气缸OUT	变更 移载垂移气缸OUT*)
DO_[54,2] 	 (	ON:= , 	OFF:= , 	LINK=>WPI_2[1,2] ,	VALUE:= arPackCylinder[14].o.ValveIn		);	(*	移载无杆气缸IN	*)
DO_[54,3] 	 (	ON:= , 	OFF:= , 	LINK=>WPI_2[1,3] ,	VALUE:= arPackCylinder[14].o.ValveOut		);	(*	移载无杆气缸OUT	*)
DO_[54,4] 	 (	ON:= , 	OFF:= , 	LINK=>WPI_2[1,4] ,	VALUE:= arPackCylinder[15].o.ValveIn		);	(*	料板支撑气缸IN	*)
DO_[54,5] 	 (	ON:= , 	OFF:= , 	LINK=>WPI_2[1,5] ,	VALUE:= arPackCylinder[15].o.ValveOut		);	(*	料板支撑气缸OUT	*)
DO_[54,6] 	 (	ON:= , 	OFF:= , 	LINK=>WPI_2[1,6] ,	VALUE:= arPackCylinder[13].o.ValveIn		);	(*	移载垂移气缸IN 变更 单排旋转气缸OUT*)
DO_[54,7] 	 (	ON:= , 	OFF:= , 	LINK=>WPI_2[1,7] ,	VALUE:= arPackCylinder[13].o.ValveOut		);	(*	移载垂移气缸OUT 变更 单排旋转气缸OUT	*)
DO_[54,8] 	 (	ON:= , 	OFF:= , 	LINK=>WPI_2[1,8] ,	VALUE:= arPackCylinder[41].o.ValveIn		);	(*  铝杯检测气缸IN	*)
DO_[55,1] 	 (	ON:= , 	OFF:= , 	LINK=>WPI_2[2,1] ,	VALUE:= arPackCylinder[41].o.ValveOut		);	(*  铝杯检测气缸OUT	*)
DO_[55,2] 	 (	ON:= , 	OFF:= , 	LINK=>WPI_2[2,2] ,	VALUE:= 		);	(*	    *)
DO_[55,3] 	 (	ON:= , 	OFF:= , 	LINK=>WPI_2[2,3] ,	VALUE:= 		);	(*		*)
DO_[55,4] 	 (	ON:= , 	OFF:= , 	LINK=>WPI_2[2,4] ,	VALUE:= 		);	(*		*)
DO_[55,5] 	 (	ON:= , 	OFF:= , 	LINK=>WPI_2[2,5] ,	VALUE:= 		);	(*		*)
DO_[55,6] 	 (	ON:= , 	OFF:= , 	LINK=>WPI_2[2,6] ,	VALUE:= 		);	(*		*)
DO_[55,7] 	 (	ON:= , 	OFF:= , 	LINK=>WPI_2[2,7] ,	VALUE:= 		);	(*		*)
DO_[55,8] 	 (	ON:= , 	OFF:= , 	LINK=>WPI_2[2,8] ,	VALUE:= 		);	(*		*)
DO_[56,1] 	 (	ON:= , 	OFF:= , 	LINK=>WPI_2[3,1] ,	VALUE:= 		);	(*		*)
DO_[56,2] 	 (	ON:= , 	OFF:= , 	LINK=>WPI_2[3,2] ,	VALUE:= 		);	(*		*)
DO_[56,3] 	 (	ON:= , 	OFF:= , 	LINK=>WPI_2[3,3] ,	VALUE:= 		);	(*		*)
DO_[56,4] 	 (	ON:= , 	OFF:= , 	LINK=>WPI_2[3,4] ,	VALUE:= 		);	(*		*)
DO_[56,5] 	 (	ON:= , 	OFF:= , 	LINK=>WPI_2[3,5] ,	VALUE:= 		);	(*		*)
DO_[56,6] 	 (	ON:= , 	OFF:= , 	LINK=>WPI_2[3,6] ,	VALUE:= 		);	(*		*)
DO_[56,7] 	 (	ON:= , 	OFF:= , 	LINK=>WPI_2[3,7] ,	VALUE:= 		);	(*		*)
DO_[56,8] 	 (	ON:= , 	OFF:= , 	LINK=>WPI_2[3,8] ,	VALUE:= 		);	(*		*)
DO_[57,1] 	 (	ON:= , 	OFF:= , 	LINK=>WPI_2[4,1] ,	VALUE:= 		);	(*		*)
DO_[57,2] 	 (	ON:= , 	OFF:= , 	LINK=>WPI_2[4,2] ,	VALUE:= 		);	(*		*)
DO_[57,3] 	 (	ON:= , 	OFF:= , 	LINK=>WPI_2[4,3] ,	VALUE:= 		);	(*		*)
DO_[57,4] 	 (	ON:= , 	OFF:= , 	LINK=>WPI_2[4,4] ,	VALUE:= 		);	(*		*)
DO_[57,5] 	 (	ON:= , 	OFF:= , 	LINK=>WPI_2[4,5] ,	VALUE:= 		);	(*		*)
DO_[57,6] 	 (	ON:= , 	OFF:= , 	LINK=>WPI_2[4,6] ,	VALUE:= 		);	(*		*)
DO_[57,7] 	 (	ON:= , 	OFF:= , 	LINK=>WPI_2[4,7] ,	VALUE:= 		);	(*		*)
DO_[57,8] 	 (	ON:= , 	OFF:= , 	LINK=>WPI_2[4,8] ,	VALUE:= 		);	(*		*)


{endregion}
END_ACTION

END_PROGRAM

// ---- POUs/MG/MotionControl.TcPOU
PROGRAM MotionControl
VAR

	arAOI_RealAxisAdmin: ARRAY[1..64] OF AOI_AxisAdmin;
	arAOI_VirtualAxisAdmin: ARRAY[1..64] OF AOI_AxisAdmin;
	arAOI_MS300Admin: ARRAY[1..1] OF AOI_MS300Admin;
	i: INT;
	MC_CamIn_Follower1: MC_CamIn;
	lrSlaveOffset: LREAL;
	lrMasterOffset: LREAL;
	MC_CamOut_Follower1: mc_camOUT;
	iCamID: MC_CAM_ID:=1;

	MC_CamTableSelect_Follower1: MC_CamTableSelect;
	CamTableFollower1: MC_CAM_REF;
	CamTableIDFollower1: MC_CAM_ID;
	table1: ARRAY[1..2] OF MC_MotionFunctionPoint; (*用于定义电子凸轮表中的关键点*)
	MC_CamIn_Follower2: MC_CamIn;
	MC_CamOut_Follower2: mc_camOUT;
	MC_CamTableSelect_Follower2: MC_CamTableSelect;
	iCamIDFollower2: MC_CAM_ID;
	iCamID2: MC_CAM_ID:=2;
	iCamID1: MC_CAM_ID:=1;
	MC_CamIn_Follower3: MC_CamIn;
	iCamID3: MC_CAM_ID;
	MC_CamOut_Follower3: mc_camOUT;
	MC_CamTableSelect_Follower3: MC_CamTableSelect;
	
	Vis_VirtualAxisRef:REFERENCE TO  UDT_AXisadmin;
	Vis_VirtualAxisNoRef: INT:=1;
	Vis_RealAxisRef:REFERENCE TO UDT_AXisadmin;
	Vis_RealAxisNoRef: INT:=1;
	xtest: BOOL;
	j: INT;
	rtestSpeed: LREAL;
	rSeepView: LREAL;
	btesetEnble: BOOL;
	bTesetMoveAbs: BOOL;
END_VAR

FOR i:=1 TO 64 DO 
	arAOI_RealAxisAdmin[i](Admin:= arRealAxisAdmin[i],enable:=HMI_AxisView[i].Enable,JogN:=HMI_AxisView[i].JogN,jogP:=HMI_AxisView[i].JogP
    ,MoveAbsolute:=HMI_AxisView[i].MoveAbs,MoveRealtive:=HMI_AxisView[i].MoveReal);
	arAOI_VirtualAxisAdmin[i](Admin:= arVirtualAxisAdmin[i]);
	arRealAxisAdmin[i].i.JogVel:=30;
	
	HMI_AxisView[i].ActPos:=arRealAxisAdmin[i].o.ActPos;
	HMI_AxisView[i].Homed:=arRealAxisAdmin[i].o.Homed;
	HMI_AxisView[i].Active:=NOT arRealAxisAdmin[i].o.StandStill;
END_FOR

Vis_RealAxisRef REF= arRealAxisAdmin[Vis_RealAxisNoRef];
Vis_VirtualAxisRef REF= arVirtualAxisAdmin[Vis_VirtualAxisNoRef];

arAOI_MS300Admin[1](admin:= arMS300Admin[1]);


TestBelt();

ACTION TestBelt:
arVirtualAxisAdmin[2].i.Vel:=rtestSpeed;
arVirtualAxisAdmin[2].i.Acc:=20000;
arVirtualAxisAdmin[2].i.Dec:=20000;
arVirtualAxisAdmin[2].i.Pos:=3300;
rSeepView:=arVirtualAxisAdmin[2].o.ActVel;
arVirtualAxisAdmin[2].i.Enable:=btesetEnble;
arVirtualAxisAdmin[2].i.MoveAbs:=bTesetMoveAbs;
END_ACTION

END_PROGRAM

// ---- Add-On-Instructions/AOI_AxisAdmin.TcPOU
FUNCTION_BLOCK AOI_AxisAdmin
VAR_INPUT
    Enable: BOOL;
	JogN: BOOL;
	JogP: BOOL;
	MoveAbsolute: BOOL;
	MoveRealtive: BOOL;
END_VAR
VAR_OUTPUT
END_VAR
VAR
	MC_Power_Axis: MC_Power;
	MC_Home_Axis: MC_Home;
	MC_MoveAbsolute_Axis: MC_MoveAbsolute;
	MC_MoveAdditive_Axis: MC_MoveAdditive;
	MC_Jog_Axis: MC_Jog;
	MC_Reset_Axis: MC_Reset;
	MC_MoveVelocity_Axis: MC_MoveVelocity;
	MC_Stop_Axis: MC_Stop;
	MC_ReadActualPosition_Axis: MC_ReadActualPosition;
	MC_SetPosition_Axis: MC_SetPosition;
	MC_MoveHome: MC_MoveAbsolute;
	R_TRIG_Home: R_TRIG;
	F_TRIG_Home: F_TRIG;
	MC_CamOut_Axis: MC_CamOut;;
	MC_Power_Stop: MC_Stop;
	MC_GearOut_Axis: mc_gearout;
	MC_MoveRelative_Axis: MC_MoveRelative;
	
	i: INT;
END_VAR
VAR_IN_OUT
	Admin: UDT_AxisAdmin;
END_VAR

IF admin.i.Disable THEN
   Disable();   
END_IF
IF admin.i.mode=0 THEN
   Enable:=FALSE;
   JogN:=FALSE;
   JogP:=FALSE;
   MoveAbsolute:=FALSE;
   MoveRealtive:=FALSE;
END_IF

Homing();
Jog();
MoveAbs();
MoveAdd();
MoveReal();
PowerOn();
Reset();
SetPos();
Stop();
Cam();
admin.o.Active:=MC_MoveAbsolute_Axis.Active OR MC_MoveAdditive_Axis.Active;
IF NOT admin.i.MoveAbs  AND NOT admin.i.MoveAdd AND NOT admin.i.MoveReal THEN
	admin.o.CmdDone:=FALSE;
END_IF
admin.Axis.ReadStatus();
admin.o.Homed:=admin.Axis.Status.Homed;
admin.o.ActPos:=admin.Axis.NcToPlc.ActPos;
admin.o.ActModuloPos:=admin.Axis.NcToPlc.ModuloActPos;
admin.o.ActVel:=admin.Axis.NcToPlc.ActVelo;
admin.o.ActTorq:=admin.Axis.NcToPlc.ActTorque;
admin.o.ErrorID:=admin.Axis.NcToPlc.ErrorCode;

admin.o.InSync:=admin.axis.Status.Coupled;
admin.o.StandStill:=admin.axis.Status.NotMoving;
admin.o.PowerOn:=admin.axis.NcToPlc.StateDWord.20;

IF admin.Axis.Status.Error  OR MC_MoveAbsolute_Axis.Error OR MC_MoveAdditive_Axis.Error OR MC_Jog_Axis.Error OR MC_MoveVelocity_Axis.Error
OR MC_MoveHome.Error OR MC_CamOut_Axis.Error OR MC_Power_Stop.Error OR MC_GearOut_Axis.Error OR MC_MoveRelative_Axis.Error  THEN
   admin.o.Error:=TRUE;
END_IF
IF admin.i.Reset THEN
   admin.o.Error:=FALSE; 
END_IF

FOR i:=1 TO 8 DO
	IF  admin.i.PosRangeTable[i][1] < admin.Axis.NcToPlc.ModuloActPos AND
        admin.Axis.NcToPlc.ModuloActPos < admin.i.PosRangeTable[i][2] THEN
		admin.o.PosInRange[i]:=TRUE;
		ELSE	
		admin.o.PosInRange[i]:=FALSE;
	END_IF
END_FOR

ACTION Cam:
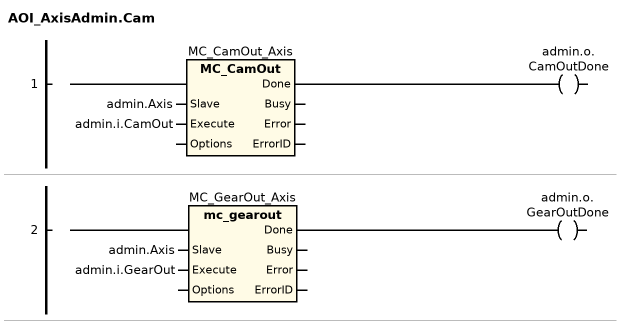
// NETWORK 1
MC_CamOut_Axis(Slave := admin.Axis, Execute := admin.i.CamOut); // MC_CamOut
admin.o.CamOutDone := MC_CamOut_Axis.Done;

// NETWORK 2
MC_GearOut_Axis(Slave := admin.Axis, Execute := admin.i.GearOut); // mc_gearout
admin.o.GearOutDone := MC_GearOut_Axis.Done;
END_ACTION

ACTION Disable:
Admin.i.CamIn:=FALSE;
Admin.i.CamOut:=FALSE;
Admin.i.Enable:=FALSE;
Admin.i.GearIn:=FALSE;
Admin.i.GearOut:=FALSE;
Admin.i.MoveAbs:=FALSE;
Admin.i.MoveAdd:=FALSE;
Admin.i.MoveVel:=FALSE;
Admin.i.JogN:=FALSE;
Admin.i.JogP:=FALSE;
Admin.i.Stop:=FALSE;
Admin.i.Home:=FALSE;
Admin.i.Reset:=FALSE;
Admin.i.SelectCamTable:=FALSE;
Admin.i.SetPosExe:=FALSE;
Admin.i.Disable:=FALSE;
Admin.i.MoveReal:=FALSE;
END_ACTION

ACTION Homing:
IF admin.i.HomeMode=0 OR admin.i.HomeMode=1 THEN
	MC_Home_Axis.HomingMode:=MC_DefaultHoming;
END_IF

IF admin.i.HomeMode=2  THEN
   MC_Home_Axis.HomingMode:=MC_Direct;
END_IF

MC_Home_Axis(
	Axis:=Admin.Axis , 
	Execute:=admin.i.Home AND admin.o.PowerOn , 
	Position:=admin.i.HomeOffset , 
	HomingMode:= , 
	BufferMode:= , 
	Options:= , 
	bCalibrationCam:= admin.i.HomeCali, 
	Done=> admin.o.HomeDone, 
	Busy=> , 
	Active=> , 
	CommandAborted=> , 
	Error=> , 
	ErrorID=> );
END_ACTION

ACTION Jog:
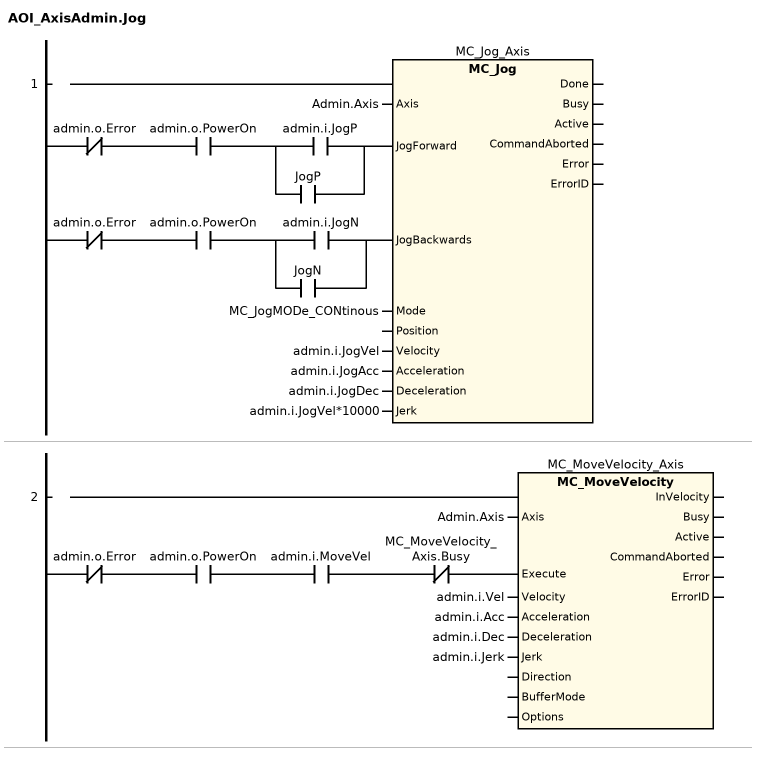
// NETWORK 1
MC_Jog_Axis(
    Axis := Admin.Axis,
    JogForward := NOT admin.o.Error AND admin.o.PowerOn AND (admin.i.JogP OR JogP),
    JogBackwards := NOT admin.o.Error AND admin.o.PowerOn AND (admin.i.JogN OR JogN),
    Mode := MC_JogMODe_CONtinous,
    Velocity := admin.i.JogVel,
    Acceleration := admin.i.JogAcc,
    Deceleration := admin.i.JogDec,
    Jerk := admin.i.JogVel*10000); // MC_Jog

// NETWORK 2
MC_MoveVelocity_Axis(
    Axis := Admin.Axis,
    Execute := NOT admin.o.Error AND admin.o.PowerOn AND admin.i.MoveVel AND NOT MC_MoveVelocity_Axis.Busy,
    Velocity := admin.i.Vel,
    Acceleration := admin.i.Acc,
    Deceleration := admin.i.Dec,
    Jerk := admin.i.Jerk); // MC_MoveVelocity
END_ACTION

ACTION MoveAbs:
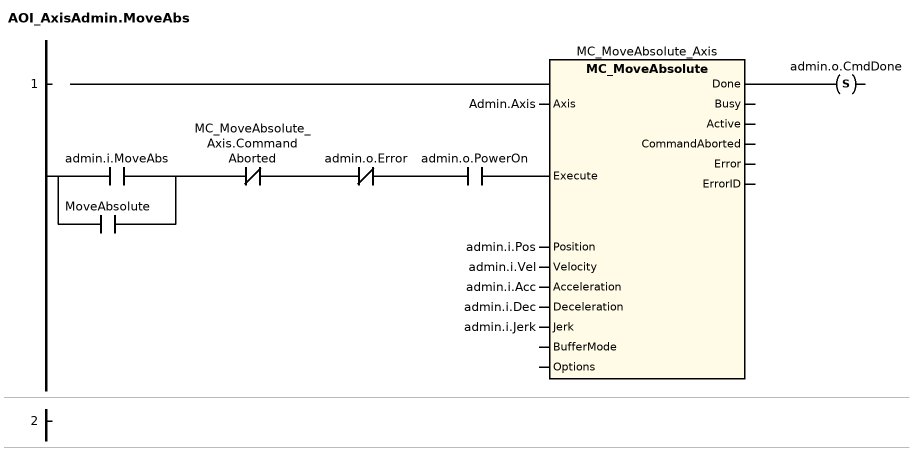
// NETWORK 1
MC_MoveAbsolute_Axis(
    Axis := Admin.Axis,
    Execute := (admin.i.MoveAbs OR MoveAbsolute) AND NOT MC_MoveAbsolute_Axis.CommandAborted AND NOT admin.o.Error AND admin.o.PowerOn,
    Position := admin.i.Pos,
    Velocity := admin.i.Vel,
    Acceleration := admin.i.Acc,
    Deceleration := admin.i.Dec,
    Jerk := admin.i.Jerk); // MC_MoveAbsolute
admin.o.CmdDone S= MC_MoveAbsolute_Axis.Done;

// NETWORK 2
END_ACTION

ACTION MoveAdd:
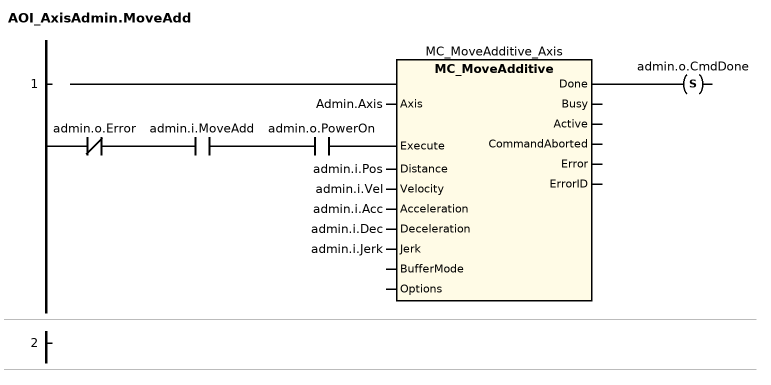
// NETWORK 1
MC_MoveAdditive_Axis(
    Axis := Admin.Axis,
    Execute := NOT admin.o.Error AND admin.i.MoveAdd AND admin.o.PowerOn,
    Distance := admin.i.Pos,
    Velocity := admin.i.Vel,
    Acceleration := admin.i.Acc,
    Deceleration := admin.i.Dec,
    Jerk := admin.i.Jerk); // MC_MoveAdditive
admin.o.CmdDone S= MC_MoveAdditive_Axis.Done;

// NETWORK 2
END_ACTION

ACTION MoveReal:
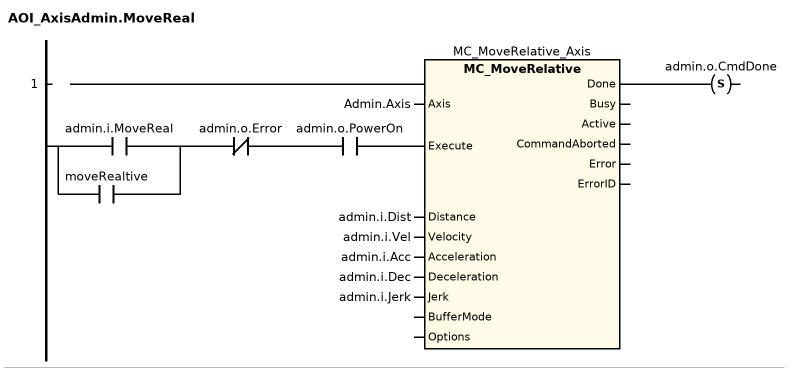
// NETWORK 1
MC_MoveRelative_Axis(
    Axis := Admin.Axis,
    Execute := (admin.i.MoveReal OR moveRealtive) AND NOT admin.o.Error AND admin.o.PowerOn,
    Distance := admin.i.Dist,
    Velocity := admin.i.Vel,
    Acceleration := admin.i.Acc,
    Deceleration := admin.i.Dec,
    Jerk := admin.i.Jerk); // MC_MoveRelative
admin.o.CmdDone S= MC_MoveRelative_Axis.Done;
END_ACTION

ACTION PowerOn:
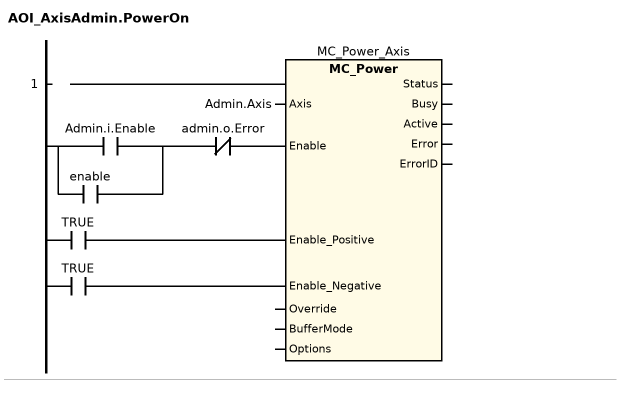
// NETWORK 1
MC_Power_Axis(
    Axis := Admin.Axis,
    Enable := (Admin.i.Enable OR enable) AND NOT admin.o.Error,
    Enable_Positive := TRUE,
    Enable_Negative := TRUE); // MC_Power
END_ACTION

ACTION Reset:
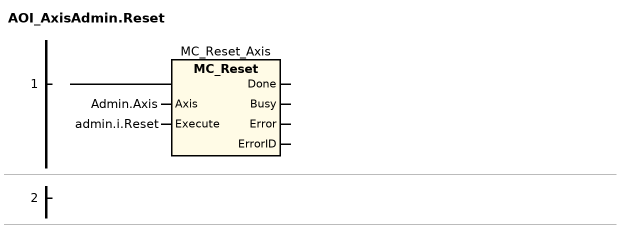
// NETWORK 1
MC_Reset_Axis(Axis := Admin.Axis, Execute := admin.i.Reset); // MC_Reset

// NETWORK 2
END_ACTION

ACTION SetPos:
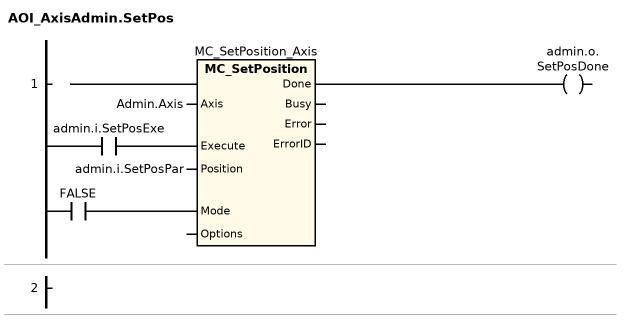
// NETWORK 1
MC_SetPosition_Axis(
    Axis := Admin.Axis,
    Execute := admin.i.SetPosExe,
    Position := admin.i.SetPosPar,
    Mode := FALSE); // MC_SetPosition
admin.o.SetPosDone := MC_SetPosition_Axis.Done;

// NETWORK 2
END_ACTION

ACTION Stop:
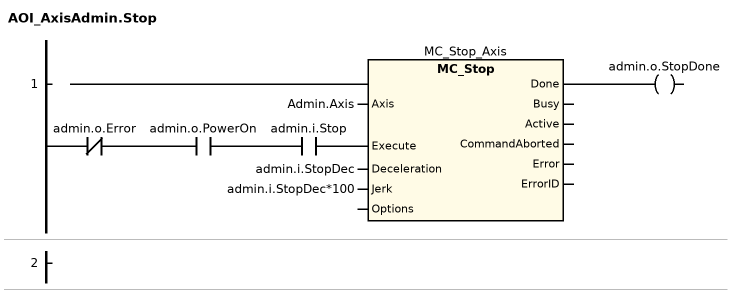
// NETWORK 1
MC_Stop_Axis(
    Axis := Admin.Axis,
    Execute := NOT admin.o.Error AND admin.o.PowerOn AND admin.i.Stop,
    Deceleration := admin.i.StopDec,
    Jerk := admin.i.StopDec*100); // MC_Stop
admin.o.StopDone := MC_Stop_Axis.Done;

// NETWORK 2
END_ACTION

END_FUNCTION_BLOCK

// ---- Add-On-Instructions/AOI_MS300Admin.TcPOU
FUNCTION_BLOCK AOI_MS300Admin
VAR_INPUT
END_VAR
VAR_OUTPUT
END_VAR
VAR
	iSeq: INT;
END_VAR
VAR_IN_OUT
 admin: UDT_MS300Admin;
END_VAR

admin.MS300.ControlWord.0:=admin.i.SwitchOn;
admin.MS300.ControlWord.1:=admin.i.EnableVoltage;
admin.MS300.ControlWord.2:=admin.i.QuickStop;
admin.MS300.ControlWord.3:=admin.i.EnableOp;
admin.MS300.ControlWord.7:=admin.i.FaultReset;
admin.MS300.ControlWord.8:=admin.i.Halt;



IF admin.i.Start AND admin.o.OperationEnable  THEN
	admin.MS300.ControlWord.4:=TRUE;
	admin.MS300.ControlWord.5:=TRUE;
	admin.MS300.ControlWord.6:=TRUE;
	ELSE
	admin.MS300.ControlWord.4:=FALSE;
	admin.MS300.ControlWord.5:=FALSE;
	admin.MS300.ControlWord.6:=FALSE;
END_IF



admin.MS300.TargetVelo:=admin.i.Vel;

admin.o.ReadyToSwitchOn:=admin.MS300.StatusWord.0;
admin.o.SwitchOn:=admin.MS300.StatusWord.1;
admin.o.OperationEnable:=admin.MS300.StatusWord.2;
admin.o.Fault:=admin.MS300.StatusWord.3;
admin.o.VoltageEnable:=admin.MS300.StatusWord.4;
admin.o.QuickStop:=admin.MS300.StatusWord.5;
admin.o.SwitchOndisabled:=admin.MS300.StatusWord.6;
admin.o.Warning:=admin.MS300.StatusWord.7;
admin.o.Reserved:=admin.MS300.StatusWord.8;
admin.o.Remote:=admin.MS300.StatusWord.9;
admin.o.TargetReached:=admin.MS300.StatusWord.10;
admin.o.InternalLimitActive:=admin.MS300.StatusWord.11;
admin.o.Operation:=admin.MS300.StatusWord.12;



CASE iSeq OF 
	0: IF admin.i.Enable THEN
		  iSeq:=10;
	   END_IF
	10:
       IF admin.o.SwitchOndisabled THEN
		  admin.i.QuickStop:=TRUE;
		  admin.i.EnableVoltage:=TRUE;
	   END_IF
	   	  iSeq:=20;
    20:
	   IF admin.o.ReadyToSwitchOn THEN
		  admin.i.SwitchOn:=TRUE;
		  admin.i.QuickStop:=TRUE;
		  admin.i.EnableVoltage:=TRUE;
		  iSeq:=30;
	   END_IF
	   	 
	30:  
	   IF admin.o.SwitchOn THEN
		  admin.i.SwitchOn:=TRUE;
		  admin.i.QuickStop:=TRUE;
		  admin.i.EnableVoltage:=TRUE;
		  admin.i.EnableOp:=TRUE;
		  iSeq:=40;
	   END_IF
	    
	40:
       IF NOT admin.i.Enable THEN
		  admin.i.SwitchOn:=FALSE;
		  admin.i.QuickStop:=FALSE;
		  admin.i.EnableVoltage:=FALSE;
		  admin.i.EnableOp:=FALSE; 
		  iSeq:=0;
	   END_IF
END_CASE


IF admin.o.Fault THEN
   iSeq:=0;
END_IF

END_FUNCTION_BLOCK

// ---- POUs/PackMaL_UN01/UN01.TcPOU
PROGRAM UN01
VAR
	Ref_Unit: REFERENCE TO UDT_UnitAdmin;
	Ref_MachineStateModel: REFERENCE TO PackMlv3_StateModel;
	ref_Master1: REFERENCE TO UDT_AXISADMIN;	
	Cfg_ModeNames: ARRAY[0..31] OF STRING;
	Cfg_DisableStates: ARRAY [0..31] OF DINT;
	Cfg_ModeTransitions: ARRAY [0..31] OF DINT;
	HMI_O_StateCurrentName: STRING(255);
	HMI_O_ModeCurrentName: STRING(255);
	iHmiErr: INT;
	Loc_diEM_AbortingDone: DINT;
	Loc_diEM_ClearingDone: DINT;
	Loc_diEM_HoldingDone: DINT;
	Loc_diEM_ResettingDone: DINT;
	Loc_diEM_StartingDone: DINT;
	Loc_diEM_StoppingDone: DINT;
	Loc_diEM_SuspendingDone: DINT;
	Loc_diEM_UnSuspendingDone: DINT;
	Loc_diEM_UnHoldingDone: DINT;	
	Loc_diEM_Fault: DINT;
	Loc_diEM_Warning: DINT;	

	// 安全复位
	tonSafetyReset: TON;
	ft_SafetyReset: F_TRIG;
	iSafetyResetSeq: INT;	
	//EtherCat	
	iFaultClearSeq: INT;
	tonFaultClear: Ton;
	bClearAllFault: BOOL;
	xDebugReset: BOOL;
	arEventEmpty: ARRAY[1..256] OF BOOL;
	arSys1EventEmpty: ARRAY[1..20] OF BOOL;
	arSys2EventEmpty: ARRAY[21..40] OF BOOL;
	arSys3EventEmpty: ARRAY[1..20] OF BOOL;	
	loc_bAnyStopError: BOOL;
	j: INT;

	tonTimeHigh: TON;
	tonTimeLow: TON;
	arBlink: ARRAY[1..10] OF blink;
	
	tonFaultHandler: Ton;	
	StopEvent: ARRAY[0..40] OF UDT_EVENT;	
	arCylinder_AOI: ARRAY[1..80] OF AOI_CylinderAdmin;	
	arVacuum_AOI: ARRAY[1..60] OF AOI_VacuumAdmin;
    arSensor_AOI: ARRAY[1..60] OF AOI_Sensoradmin;	
	arHeat_AOI: ARRAY[1..8] OF Aoi_HeatBase;
    bUnitFS: BOOL;

	diUnitStopEvent0: DINT;
	rtWorkLocMode: R_trig;
	iRecipeSeq: INT;
	tonCmdReset: TON;
	tonCmdStart: TON;
	diSys1StopEvent1: DINT;
	diSys1StopEvent2: DINT;
	diSys2StopEvent1: DINT;
	diSys2StopEvent2: DINT;
	diSys3StopEvent1: DINT;
	diSys3StopEvent2: DINT;
	diSys3StopEvent3: DINT;
	rtAllaxisHomed: R_TRIG;
	tonRecipeSeq: Ton;
	
	tongeneralEvent0:ARRAY[0..255] OF Ton;

	diSys3StopEvent4: DINT;
	bSys1StopError: BOOL;
	bSys2StopError: BOOL;
	bSys3StopError: BOOL;

	iC: INT;
	
	arDropCylinder_AOI: ARRAY[1..40] OF AOI_CylinderAdmin;	
	iNotDone: INT;
	aoiActiveTotalTime: AOI_Timer;
	aoiWorkTotalTime: AOI_Timer;
	aoi10MinuteTime: AOI_Timer;
	
	rtGoodCount: R_TRIG;
	rtNoGoodCount: R_trig;
	rMaxCounterTime: DINT;
	rMaxDropTime: DINT;
	i: INT;
	iInitCnt: INT;
	iAutoCut: INT;
	tonAutoCut: Ton;
	iCutCnt: INT;
	bBoxRecipeUpdate: BOOL;
	bEn10Minute: BOOL;
	bReset10Minute: BOOL;
	diTransferCntOld: DINT;
	tonRecipeReset: Ton;
	bFirstCyclinderScan: BOOL;
	bAnySaftyDoorOpen: BOOL;
	tonCounterAirOpen: Ton;
END_VAR

VAR CONSTANT
   EM_OK: ARRAY[0..64] OF BOOL :=[65(0)];
   diEm_Done: DINT:=0;
END_VAR

//PLC IP地址IP 192.168.1.10 HMI1 IP 192.168.1.12 HMI2 IP 192.168.1.13 路由器 密码IPB19021 账号admin 
//激光打标机IP 192.168.1.20 
Ref_Unit REF=Unit01;
Ref_MachineStateModel REF= UN01_MachineStateModel;
ref_Master1 REF= arVirtualAxisAdmin[1];
CM02_ConditionsModules();
CM03_Cylinder();
CM04_Vacuum();
CM05_Sensor();
CM06_Heat();
CM07_Counters();
CM10_LightStatus();
SR02_Recipe();
UP01_PackML();
UP02_StateComplete();
EM01_Master();
EM02_Follower1();
EM03_Follower2();
EM04_FOllower3();
EM05_Counters();
EM06_Follower4_5();
EM07_Belt6();
EM08_Belt7();
SR91_OEE();
CM01_OperationLocal();
SR05_Manual();

IF NOT bUnitFS THEN
   SR01_Initialize();
END_IF

SR03_FaultHandler();
SR04_Parameter();
SR90_SafetyReset();
SR99_FaultClear();

DebugPro();

ACTION CM01_OperationLocal:
Ref_MachineStateModel.Cmd_Clear:=HMI_LocModeInput.ClearFault OR xDebugReset;
bAnySaftyDoorOpen:=arSafeDoorSts[19] OR arSafeDoorSts[20] OR arSafeDoorSts[21] OR arSafeDoorSts[22];
//前后设备急停串联
IF (glb_diEstopButton_UN01<>0) THEN
	Ref_MachineStateModel.Cmd_Abort:=TRUE;
	glb_AllAxisHomed_UN01:=FALSE;
	ELSE
	Ref_MachineStateModel.Cmd_Abort:=FALSE;
END_IF
//清除故障
IF Ref_MachineStateModel.Cmd_Clear THEN
   bClearAllFault:=TRUE;
END_IF
//停机
IF (HMI_LocModeInput.Stop OR glb_bStopButton_UN01) OR 
   (bAnySaftyDoorOpen AND Ref_MachineStateModel.Sts_Resetting) AND NOT Ref_MachineStateModel.Sts_Held THEN
	Ref_MachineStateModel.Cmd_Stop:=TRUE;
	ELSE
	Ref_MachineStateModel.Cmd_Stop:=FALSE;	
END_IF
//暂停
IF ((loc_bAnyStopError OR bAnySaftyDoorOpen) AND Ref_MachineStateModel.Sts_Execute) 
OR HMI_LocModeInput.Hold THEN
	Ref_MachineStateModel.Cmd_Hold:=TRUE;
	ELSE
	Ref_MachineStateModel.Cmd_Hold:=FALSE;	
END_IF
//启动
tonCmdStart(IN:= (HMI_LocModeInput.Start OR glb_bStartButton_UN01), PT:=T#2S , Q=> , ET=> );
IF tonCmdStart.Q AND glb_bAllSafetyOk 
AND NOT loc_bAnyStopError  
AND Ref_MachineStateModel.Sts_Idle
AND glb_bModeSwitch_UN01 THEN
	Ref_MachineStateModel.Cmd_Start:=TRUE;
	ELSE
	Ref_MachineStateModel.Cmd_Start:=FALSE;	
END_IF
//复位
tonCmdReset(IN:= (HMI_LocModeInput.Reset OR glb_bResetButton_UN01), PT:=T#2S , Q=> , ET=> );
IF tonCmdReset.Q AND NOT loc_bAnyStopError AND glb_bModeSwitch_UN01 THEN
   IF HMI_LocModeINPUT.Reset THEN
	  glb_AllAxisHomed_UN01:=FALSE;
   END_IF
   Ref_MachineStateModel.Cmd_Reset:=TRUE;
   ELSE
   Ref_MachineStateModel.Cmd_Reset:=FALSE;	 
END_IF

//安全复位
IF (glb_bResetButton_UN01 OR glb_bResetButton_UN02) AND
NOT glb_bAllSafetyOk THEN
   glb_bSafetyReset:=TRUE;
END_IF

//解除暂停
IF tonCmdStart.Q  AND Ref_MachineStateModel.Sts_Held  
AND glb_bModeSwitch_UN01 AND NOT loc_bAnyStopError THEN
	Ref_MachineStateModel.Cmd_UnHold:=TRUE;
	ELSE
    Ref_MachineStateModel.Cmd_UnHold:=FALSE;
END_IF

//等待启动
IF Ref_MachineStateModel.Sts_Idle THEN
	glb_AllAxisHomed_UN01:=TRUE;
END_IF
END_ACTION

ACTION CM02_ConditionsModules:
Loc_diEM_AbortingDone:=MEMCMP(pBuf1:=ADR(Ref_Unit.EM_Aborting_Done) , pBuf2:=ADR(Ref_Unit.EM_Selected) , n:=SIZEOF(Ref_Unit.EM_Selected));
Loc_diEM_ClearingDone:=MEMCMP(pBuf1:=ADR(Ref_Unit.EM_Clearing_Done) , pBuf2:=ADR(Ref_Unit.EM_Selected) , n:=SIZEOF(Ref_Unit.EM_Selected));
Loc_diEM_HoldingDone:=MEMCMP(pBuf1:=ADR(Ref_Unit.EM_Holding_Done) , pBuf2:=ADR(Ref_Unit.EM_Selected) , n:=SIZEOF(Ref_Unit.EM_Selected));
Loc_diEM_ResettingDone:=MEMCMP(pBuf1:=ADR(Ref_Unit.EM_Resetting_Done) , pBuf2:=ADR(Ref_Unit.EM_Selected) , n:=SIZEOF(Ref_Unit.EM_Selected));
Loc_diEM_StartingDone:=MEMCMP(pBuf1:=ADR(Ref_Unit.EM_Starting_Done) , pBuf2:=ADR(Ref_Unit.EM_Selected) , n:=SIZEOF(Ref_Unit.EM_Selected));
Loc_diEM_StoppingDone:=MEMCMP(pBuf1:=ADR(Ref_Unit.EM_Stopping_Done) , pBuf2:=ADR(Ref_Unit.EM_Selected) , n:=SIZEOF(Ref_Unit.EM_Selected));
Loc_diEM_SuspendingDone:=MEMCMP(pBuf1:=ADR(Ref_Unit.EM_Suspending_Done) , pBuf2:=ADR(Ref_Unit.EM_Selected) , n:=SIZEOF(Ref_Unit.EM_Selected));
Loc_diEM_UnSuspendingDone:=MEMCMP(pBuf1:=ADR(Ref_Unit.EM_UnSuspending_Done) , pBuf2:=ADR(Ref_Unit.EM_Selected) , n:=SIZEOF(Ref_Unit.EM_Selected));
Loc_diEM_UnHoldingDone:=MEMCMP(pBuf1:=ADR(Ref_Unit.EM_UnHolding_Done) , pBuf2:=ADR(Ref_Unit.EM_Selected) , n:=SIZEOF(Ref_Unit.EM_Selected));

Loc_diEM_Fault:=MEMCMP(pBuf1:=ADR(Ref_Unit.EM_Fault) , pBuf2:=ADR(EM_OK) , n:=SIZEOF(Ref_Unit.EM_Selected));
Loc_diEM_Warning:=MEMCMP(pBuf1:=ADR(Ref_Unit.EM_Warning) , pBuf2:=ADR(EM_OK) , n:=SIZEOF(Ref_Unit.EM_Selected));

Ref_Unit.EM_Selected:=HMI_EMSelectUn01;
END_ACTION

ACTION CM03_Cylinder:
FOR i:= 1 TO 60 DO
	arPackCylinder[i].i.CheckTime:=10000;
	arPackCylinder[i].i.Mode:=1;	
    arCylinder_AOI[i](Admin:= arPackCylinder[i]);
END_FOR
	arDropBufferCyclinder[1].i.CheckTime:=10000;
	arDropBufferCyclinder[1].i.Mode:=1;
	arDropBufferCyclinder[2].i.CheckTime:=10000;
	arDropBufferCyclinder[2].i.Mode:=1;
arCylinder_AOI[61](Admin:= arDropBufferCyclinder[1]);
arCylinder_AOI[62](Admin:= arDropBufferCyclinder[2]);
IF NOT bFirstCyclinderScan THEN
   bFirstCyclinderScan:=TRUE;
END_IF
END_ACTION

ACTION CM04_Vacuum:
FOR i:=1 TO 60 DO
	arPackVacuum[i].i.CheckTime:=5000;
	arPackVacuum[i].i.BlowTime:=1000;
	arVacuum_AOI[i](admin:= arPackVacuum[i]);
END_FOR
END_ACTION

ACTION CM05_Sensor:
FOR i:=1 TO 60 DO
	arSensor_AOI[i](Admin:=arPackSensor[i] );
END_for
END_ACTION

ACTION CM06_Heat:
	arHeat_AOI[1](	Enable:=NOT HMI_HeatDisable , 	PV:=HMI_HeatTempAct[1] , 	SV:= HMI_HeatTempSet[1], 
 	Reset:= ,HighLimit:= 30,lowLimit:= 30,MaxLimit:=300,Kp:=20,Ki:=0.5,Kd:=3,
	Active=> arPackHeatRealy[1], 
	Error=> );
	arHeat_AOI[2](	Enable:=NOT HMI_HeatDisable , 	PV:=HMI_HeatTempAct[2] , 	SV:= HMI_HeatTempSet[2], 
	Reset:= ,HighLimit:= 30, lowLimit:= 30,MaxLimit:=300,Kp:=20,Ki:=0.5,Kd:=3,
	Active=> arPackHeatRealy[2], 
	Error=> );
	arHeat_AOI[3](	Enable:=NOT HMI_HeatDisable , 	PV:=HMI_HeatTempAct[3] , 	SV:= HMI_HeatTempSet[3], 
    Reset:= ,HighLimit:= 30, lowLimit:= 30,MaxLimit:=300,Kp:=20,Ki:=0.5,Kd:=3,
	Active=> arPackHeatRealy[3], 
	Error=> );
	arHeat_AOI[4](	Enable:=NOT HMI_HeatDisable , 	PV:=HMI_HeatTempAct[4] , 	SV:= HMI_HeatTempSet[4], 
    Reset:= ,HighLimit:= 30, lowLimit:= 30,MaxLimit:=300,Kp:=20,Ki:=0.5,Kd:=3,		
	Active=> arPackHeatRealy[4], 
	Error=> );
	arHeat_AOI[5](	Enable:=NOT HMI_HeatDisable , 	PV:=HMI_HeatTempAct[5] , 	SV:= HMI_HeatTempSet[5], 
    Reset:= ,HighLimit:= 30, lowLimit:= 30,MaxLimit:=300,Kp:=20,Ki:=0.5,Kd:=3,		
	Active=> arPackHeatRealy[5], 
	Error=> );
	arHeat_AOI[6](	Enable:=NOT HMI_HeatDisable , 	PV:=HMI_HeatTempAct[6] , 	SV:= HMI_HeatTempSet[6],
    Reset:= ,HighLimit:= 30, lowLimit:= 30,MaxLimit:=300,Kp:=20,Ki:=0.5,Kd:=3, 
	Active=> arPackHeatRealy[6], 
	Error=> );
	arHeat_AOI[7](	Enable:=NOT HMI_HeatDisable , 	PV:=HMI_HeatTempAct[7] , 	SV:= HMI_HeatTempSet[7],
    Reset:= ,HighLimit:= 30, lowLimit:= 30,MaxLimit:=300,Kp:=20,Ki:=0.5,Kd:=3, 
	Active=> arPackHeatRealy[7], 
	Error=> );
	arHeat_AOI[8](	Enable:=NOT HMI_HeatDisable , 	PV:=HMI_HeatTempAct[8] , 	SV:= HMI_HeatTempSet[8],
    Reset:= ,HighLimit:= 30, lowLimit:= 30,MaxLimit:=300,Kp:=20,Ki:=0.5,Kd:=3, 
	Active=> arPackHeatRealy[8], 
	Error=> );	
	
	HMI_HeatTempAct[1]:=INT_TO_REAL(EL3312[1,1].Value)/10;
	HMI_HeatTempAct[2]:=INT_TO_REAL(EL3312[1,2].Value)/10;
	HMI_HeatTempAct[3]:=INT_TO_REAL(EL3312[2,1].Value)/10;
	HMI_HeatTempAct[4]:=INT_TO_REAL(EL3312[2,2].Value)/10;
	HMI_HeatTempAct[5]:=INT_TO_REAL(EL3312[3,1].Value)/10;
	HMI_HeatTempAct[6]:=INT_TO_REAL(EL3312[3,2].Value)/10;   
	HMI_HeatTempAct[7]:=INT_TO_REAL(EL3312[4,1].Value)/10;
	HMI_HeatTempAct[8]:=INT_TO_REAL(EL3312[4,2].Value)/10;
END_ACTION

ACTION CM07_Counters:
iInitCnt:=0;
rMaxDropTime:=0;
rMaxCounterTime:=0;
FOR ic:=1 TO 10 DO
	arCounters[iC](
		In_Total:= RecipeBuffer.amount, 
		Quantity:= RecipeBuffer.Counters[iC].Quantity, 
		ProcessTime=> HMI_OEEView.CounterProcessTime[iC] ,
		Axis:= arRealAxisAdmin[iC], 
		Checktime:= HMI_CntCheckTime,
		DropSensor:= arDropSensor[iC], 
		LowSensor:= arLowSensor[iC], 
		HighSensor:= arhighSensor[iC],
		DropFlag:= glb_BinBelt1.bin[iC].arDrop[iC],
		Cylinder:= arDropCylinder[iC]);	
END_FOR
FOR ic:=11 TO 20 DO
	arCounters[iC](
		In_Total:= RecipeBuffer.amount, 
		Quantity:= RecipeBuffer.Counters[iC].Quantity,
       	CheckTime:= 1500,
		ProcessTime=> HMI_OEEView.CounterProcessTime[iC] ,
		Axis:= arRealAxisAdmin[iC], 
		Checktime:= HMI_CntCheckTime,
		DropSensor:= arDropSensor[iC], 
		LowSensor:= arLowSensor[iC], 
		HighSensor:= arhighSensor[iC],
		DropFlag:= glb_BinBelt1.bin[iC+20].arDrop[iC+20],
		Cylinder:= arDropCylinder[iC]);	
END_FOR

FOR ic:=21 TO 30 DO
	arCounters[iC](
		In_Total:= RecipeBuffer.amount, 
		Quantity:= RecipeBuffer.Counters[iC].Quantity, 
		ProcessTime=> HMI_OEEView.CounterProcessTime[iC] ,
		Axis:= arRealAxisAdmin[iC], 
		Checktime:= HMI_CntCheckTime,
		DropSensor:= arDropSensor[iC], 
		LowSensor:= arLowSensor[iC], 
		HighSensor:= arhighSensor[iC],
		DropFlag:= glb_BinBelt2.bin[ic-20].arDrop[iC-20],
		Cylinder:= arDropCylinder[iC]);	
END_FOR

FOR ic:=31 TO 40 DO
	arCounters[iC](
		In_Total:= RecipeBuffer.amount, 
		Quantity:= RecipeBuffer.Counters[iC].Quantity, 
		ProcessTime=> HMI_OEEView.CounterProcessTime[iC] ,
		Axis:= arRealAxisAdmin[iC], 
		Checktime:= HMI_CntCheckTime,
		DropSensor:= arDropSensor[iC], 
		LowSensor:= arLowSensor[iC], 
		HighSensor:= arhighSensor[iC],
		DropFlag:= glb_BinBelt2.bin[iC].arDrop[iC],
		Cylinder:= arDropCylinder[iC]);	
END_FOR
  
FOR iC:=1 TO 40 DO
	arDropCylinder_AOI[iC](Admin:= arDropCylinder[iC]);
	arDropCylinder[iC].i.CheckTime:=1500;
	arDropCylinder[iC].i.Mode:=1;	
   IF NOT  arCounters[iC].Busy THEN
      IF rMaxCounterTime < arCounters[iC].ProcessTime THEN
		 rMaxCounterTime:= arCounters[iC].ProcessTime;
	  END_IF
   END_IF  
   arCounters[iC].SkipAlarm:=HMI_SkipCntAlarm[iC];
   arCounters[iC].CheckCnt:=HMI_CntCheck[iC];
   HMI_CountersCntUp[ic]:=arCounters[iC].CntUp;
   
   HMI_OEEView.DropProcessTime[ic]:=(arDropCylinder_AOI[iC].ActInTime+arDropCylinder_AOI[iC].ActOutTime)/2;
   IF rMaxDropTime<HMI_OEEView.DropProcessTime[ic] THEN
	  rMaxDropTime:=HMI_OEEView.DropProcessTime[ic];  
   END_IF
END_FOR
END_ACTION

ACTION CM10_LightStatus:

IF glb_bAllSafetyOk THEN
	glb_bResetBottonLight_UN01:=TRUE;
	ELSE 
    glb_bResetBottonLight_UN01:=arBlink[1].OUT;
END_IF

{region Lihgtsys1} 
//红灯
glb_arLightRed_UN01[1]:=Ref_MachineStateModel.Sts_Aborted OR Ref_MachineStateModel.Sts_Aborting OR (arblink[1].OUT AND bSys1StopError);
glb_arLightAlarm_UN01[1]:=(glb_arLightRed_UN01[1] OR glb_arLightYellow_UN01[1]) AND NOT HMI_AlarmMute;
//绿灯	  
glb_arLightGreen_UN01[1]:= Ref_MachineStateModel.Sts_Execute OR  Ref_MachineStateModel.Sts_Stopping OR
( arblink[1].OUT AND NOT bSys1StopError  AND NOT Ref_MachineStateModel.Sts_Aborted AND NOT Ref_MachineStateModel.Sts_Resetting
AND( Ref_MachineStateModel.Sts_Stopped OR Ref_MachineStateModel.Sts_Idle OR Ref_MachineStateModel.Sts_Held))
OR (Ref_MachineStateModel.Sts_Resetting  AND arblink[2].OUT);	 
//黄灯
glb_arLightYellow_UN01[1]:= (HMI_GeneralEvent[2].ID[1] OR HMI_GeneralEvent[2].ID[2] OR HMI_GeneralEvent[2].ID[3] OR HMI_GeneralEvent[2].ID[4]
OR HMI_GeneralEvent[2].ID[5] OR HMI_GeneralEvent[2].ID[6] OR HMI_GeneralEvent[2].ID[7] OR HMI_GeneralEvent[2].ID[8] OR HMI_GeneralEvent[2].ID[9]
OR HMI_GeneralEvent[2].ID[10] OR HMI_GeneralEvent[2].ID[11] OR HMI_GeneralEvent[2].ID[12] OR HMI_GeneralEvent[2].ID[13] OR HMI_GeneralEvent[2].ID[14]
OR HMI_GeneralEvent[2].ID[15] OR HMI_GeneralEvent[2].ID[16] OR HMI_GeneralEvent[2].ID[17] OR HMI_GeneralEvent[2].ID[18] OR HMI_GeneralEvent[2].ID[19]
OR HMI_GeneralEvent[2].ID[20]) AND arblink[1].OUT;	 	 
		  
(*照明灯*)  
glb_arLightRelay_UN01[1]:= arSafeDoorSts[1] OR arSafeDoorSts[2] OR arSafeDoorSts[3] OR arSafeDoorSts[4] OR
arSafeDoorSts[5] OR arSafeDoorSts[6] OR arSafeDoorSts[7] OR arSafeDoorSts[8] OR
arSafeDoorSts[9] ;
	   
{end_region}				
{region Lihgtsys2} 					 

glb_arLightRed_UN01[2]:=Ref_MachineStateModel.Sts_Aborted OR Ref_MachineStateModel.Sts_Aborted OR ( arblink[1].OUT AND bSys2StopError );
glb_arLightAlarm_UN01[2]:=(glb_arLightRed_UN01[2] OR glb_arLightYellow_UN01[2]) AND NOT HMI_AlarmMute;
		  
glb_arLightGreen_UN01[2]:= Ref_MachineStateModel.Sts_Execute OR Ref_MachineStateModel.Sts_Stopping OR
( arblink[1].OUT AND NOT bSys2StopError  AND NOT Ref_MachineStateModel.Sts_Aborted AND NOT Ref_MachineStateModel.Sts_Resetting
AND( Ref_MachineStateModel.Sts_Stopped OR Ref_MachineStateModel.Sts_Idle OR Ref_MachineStateModel.Sts_Held))
OR (Ref_MachineStateModel.Sts_Resetting  AND arblink[2].OUT);
 
//黄灯
glb_arLightYellow_UN01[2]:= (HMI_GeneralEvent[2].ID[21] OR HMI_GeneralEvent[2].ID[22] OR HMI_GeneralEvent[2].ID[23] OR HMI_GeneralEvent[2].ID[24]
OR HMI_GeneralEvent[2].ID[25] OR HMI_GeneralEvent[2].ID[26] OR HMI_GeneralEvent[2].ID[27] OR HMI_GeneralEvent[2].ID[28] OR HMI_GeneralEvent[2].ID[29]
OR HMI_GeneralEvent[2].ID[30] OR HMI_GeneralEvent[2].ID[31] OR HMI_GeneralEvent[2].ID[32] OR HMI_GeneralEvent[2].ID[33] OR HMI_GeneralEvent[2].ID[34]
OR HMI_GeneralEvent[2].ID[35] OR HMI_GeneralEvent[2].ID[36] OR HMI_GeneralEvent[2].ID[37] OR HMI_GeneralEvent[2].ID[38] OR HMI_GeneralEvent[2].ID[39]
OR HMI_GeneralEvent[2].ID[40]) AND arblink[1].OUT;		   
(*照明灯*)

glb_arLightRelay_UN01[2]:=arSafeDoorSts[10] OR arSafeDoorSts[11] OR arSafeDoorSts[12] OR arSafeDoorSts[13] OR
arSafeDoorSts[14] OR arSafeDoorSts[15] OR arSafeDoorSts[16] OR arSafeDoorSts[17] OR
arSafeDoorSts[18] ;
	  
{end_region}		   

{region Lihgtsys3} 	

glb_arLightRed_UN01[3]:=Ref_MachineStateModel.Sts_Aborted OR Ref_MachineStateModel.Sts_Aborted OR (arblink[1].OUT AND bSys3StopError);
glb_arLightAlarm_UN01[3]:=glb_arLightRed_UN01[3] AND NOT HMI_AlarmMute;
			   
							  
glb_arLightGreen_UN01[3]:= Ref_MachineStateModel.Sts_Execute OR Ref_MachineStateModel.Sts_Stopping OR
( arblink[1].OUT AND NOT bSys3StopError  AND NOT Ref_MachineStateModel.Sts_Aborted AND NOT Ref_MachineStateModel.Sts_Resetting
AND( Ref_MachineStateModel.Sts_Stopped OR Ref_MachineStateModel.Sts_Idle OR Ref_MachineStateModel.Sts_Held))
OR (Ref_MachineStateModel.Sts_Resetting  AND arblink[2].OUT);
//黄灯
glb_arLightYellow_UN01[3]:= ( HMI_GeneralEvent[0].ID[1] OR HMI_GeneralEvent[0].ID[2] ) AND arblink[1].OUT;		   
(*照明灯*)

{end_region}

arBlink[1](TimeH:=100 , TimeL:=1000 , OUT=> );
arBlink[2](TimeH:=200 , TimeL:=200 , OUT=> );
END_ACTION

ACTION SR01_Initialize:
glb_bCounterAirValve_UN01:=TRUE;
bUnitFS:=TRUE;
HMI_EMSelectUN01[1]:=TRUE;
HMI_EMSelectUN01[2]:=TRUE;
HMI_EMSelectUN01[3]:=TRUE;
HMI_EMSelectUN01[4]:=TRUE;
HMI_EMSelectUN01[5]:=TRUE;
HMI_EMSelectUN01[6]:=TRUE;
HMI_EMSelectUN01[7]:=TRUE;
HMI_EMSelectUN01[8]:=TRUE;
	
;
END_ACTION

ACTION SR02_Recipe:
rtWorkLocMode(CLK:=HMI_LocModeEnable , Q=> );
rtAllaxisHomed(CLK:= glb_AllAxisHomed_UN01, Q=> );
tonRecipeReset(IN:=glb_bResetButton_UN01 AND Ref_MachineStateModel.Sts_Execute , PT:= T#5S , Q=> , ET=> );

CASE iRecipeSeq OF 
	0: 
	   HMI_RecipeReset:=TRUE;
	   bBoxRecipeUpdate:=FALSE;
       IF  glb_AllAxisHomed_UN01  THEN
		   IF HMI_LocModeEnable THEN
			  iRecipeSeq:=10;
		   END_IF
		   IF Hmi_Input.ModifyRecipe OR tonRecipeReset.Q THEN 
			  iRecipeSeq:=20;
			  HMI_RecipeReset:=FALSE;
		   END_IF
		   IF HMI_RecipeRedo THEN
			  HMI_RecipeReset:=FALSE;
			  iRecipeSeq:=300;  
		   END_IF
		   IF HMI_RecipCancel THEN
			  HMI_RecipeReset:=FALSE;
			  iRecipeSeq:=200;  
		   END_IF
	   END_IF
	
	10:(*本地模拟生产配方*)
        Hmi_Output.InQuantity:=49;
		Hmi_Output.OutQuantity:=0;
		FOR i:=1 TO 40 DO
			Hmi_Output.Counters[i].Quantity:=5;
			Hmi_Output.Counters[i].ID:=i;
		END_FOR
	    iRecipeSeq:=90;	


     20:
        (**生产任务配方**)
		IF Hmi_Recipe.amount<>0 THEN//配方有效
			RecipeBuffer:=HMI_RECIPE;
			RecipeBuffer.user:=HMI_RECIPE.user;
			Hmi_Output.InQuantity:=RecipeBuffer.amount;
			Hmi_Output.OutQuantity:=0;
			FOR i:=1 TO 40 DO
				Hmi_Output.Counters[i].Quantity:=RecipeBuffer.Counters[i].Quantity;
				Hmi_Output.Counters[i].ID:=RecipeBuffer.Counters[i].ID;
			END_FOR
			iRecipeSeq:=90;	
		ELSE//配方无效
            iRecipeSeq:=200;	
		END_IF
 

		
	90: //复位料仓
        Glb_BinList.Reset:=TRUE;
		FOR i:=1 TO 40 DO
		    arCounters[i].Reset:=TRUE;
		END_FOR 
	    iRecipeSeq:=91;
    91: //复位数粒 		
		FOR i:=1 TO 40 DO
		    arCounters[i].Reset:=FALSE;
		END_FOR
		Glb_BinList.Reset:=FALSE;
		glb_lrMasterTargetCnt:=glb_lrMasterTargetCnt + Hmi_Output.InQuantity;
		glb_lrBelt1TargetCnt:=glb_lrBelt1TargetCnt + Hmi_Output.InQuantity + HMI_B1DropBinNo;
		glb_lrBelt2Targetcnt:=glb_lrBelt2Targetcnt + Hmi_Output.InQuantity + HMI_B2DropBinNo;
		glb_lrBelt3Targetcnt:=glb_lrBelt3Targetcnt+ Hmi_Output.InQuantity + HMI_B3DropBinNo3;	
		iRecipeSeq:=92;
		
	92:	
	    tonRecipeSeq(IN:=TRUE, PT:=T#1S , Q=> , ET=> );
		IF tonRecipeSeq.Q THEN
	       tonRecipeSeq(IN:=FALSE, PT:=T#1S , Q=> , ET=> );	
			HMI_Output.RecipeComplete:=FALSE;
			Hmi_Input.ModifyRecipe:=FALSE;
			HMI_Output.RecipeModifyDone:=TRUE;	  	  
            iRecipeSeq:=93;	
		END_IF	
		
	93:
        tonRecipeSeq(IN:=TRUE, PT:=T#1S , Q=> , ET=> );
		IF tonRecipeSeq.Q THEN
	       tonRecipeSeq(IN:=FALSE, PT:=T#1S , Q=> , ET=> );	  	  
           iRecipeSeq:=100;	
		END_IF	
	 
	100:
	    glb_BinBelt1.bin[1].Name:=RecipeBuffer.user;
		glb_BinBelt1.bin[1].Amount:=RecipeBuffer.amount;//获取生产数量
	    HMI_RecipeAbort:=FALSE;
        Hmi_Output.RecipeEmplty:=FALSE;
		IF glb_lrBelt1wrkCnt>14  AND NOT bBoxRecipeUpdate  THEN
		   glb_lrBoxTargetCnt := glb_lrBoxTargetCnt+Hmi_Output.InQuantity/7;
		   bBoxRecipeUpdate:=TRUE;
		END_IF

		IF glb_lrBelt1wrkCnt = glb_lrBelt1TargetCnt AND glb_lrBelt2wrkCnt = glb_lrBelt2TargetCnt THEN
			HMI_Output.RecipeComplete:=TRUE;
		END_IF
		
	    IF HMI_Output.RecipeComplete THEN
		   HMI_Output.RecipeModifyDone:=FALSE;
	       iRecipeSeq:=110;
		   ELSE IF NOT glb_AllAxisHomed_UN01 THEN//配方被中止
			           HMI_RecipeAbort:=TRUE;
					   iRecipeSeq:=900;
		        END_IF
		END_IF
		
    
    110:
	    tonRecipeSeq(IN:=TRUE, PT:=T#1S , Q=> , ET=> );
		IF tonRecipeSeq.Q THEN
	       tonRecipeSeq(IN:=FALSE, PT:=T#1S , Q=> , ET=> );	
           iRecipeSeq:=0;		
		END_IF
		
(***************************************************************)		
    200: 
        HMI_RecipeAbort:=FALSE;
	    tonRecipeSeq(IN:=TRUE, PT:=T#1S , Q=> , ET=> );
		IF tonRecipeSeq.Q THEN
	       tonRecipeSeq(IN:=FALSE, PT:=T#1S , Q=> , ET=> );	
			HMI_Output.RecipeComplete:=FALSE;
			Hmi_Input.ModifyRecipe:=FALSE;
			HMI_Output.RecipeModifyDone:=TRUE;	  	  
           iRecipeSeq:=210;	
		END_IF	
    210:
	    tonRecipeSeq(IN:=TRUE, PT:=T#1S , Q=> , ET=> );
		IF tonRecipeSeq.Q THEN
	       tonRecipeSeq(IN:=FALSE, PT:=T#1S , Q=> , ET=> );	
			HMI_Output.RecipeComplete:=TRUE;
			HMI_Output.RecipeModifyDone:=FALSE;	  	  
           iRecipeSeq:=220;	
		END_IF	

    220:
	    tonRecipeSeq(IN:=TRUE, PT:=T#1S , Q=> , ET=> );
		IF tonRecipeSeq.Q THEN
	       tonRecipeSeq(IN:=FALSE, PT:=T#1S , Q=> , ET=> );		  	  
           iRecipeSeq:=0;	
		END_IF	
(***********************************************************)		
	300:
		IF RecipeBuffer.amount<>0 THEN
			Hmi_Output.InQuantity:=RecipeBuffer.amount;
			Hmi_Output.OutQuantity:=0;
			FOR i:=1 TO 40 DO
				Hmi_Output.Counters[i].Quantity:=RecipeBuffer.Counters[i].Quantity;
				Hmi_Output.Counters[i].ID:=RecipeBuffer.Counters[i].ID;
			END_FOR
			iRecipeSeq:=90;	
		ELSE
            iRecipeSeq:=200;	
		END_IF	
			
	900:
	    Hmi_Output.InQuantity:=0;
		Hmi_Output.OutQuantity:=0;
		Hmi_Output.RecipeEmplty:=TRUE;
		HMI_Output.RecipeModifyDone:=FALSE;
		HMI_Output.RecipeComplete:=FALSE;

        FOR i:=1 TO 40 DO
		    arCounters[i].Reset:=TRUE;	
		END_FOR
	    Glb_BinList.Reset:=TRUE;
	 	iRecipeSeq:=1000;
	1000:
        HMI_Output.RecipeComplete:=FALSE;
		HMI_Output.RecipeModifyDone:=FALSE;	
		Glb_BinList.Reset:=FALSE;
		FOR i:=1 TO 40 DO
		    arCounters[i].Reset:=FALSE;	
		END_FOR
		
		iRecipeSeq:=0;
END_CASE
END_ACTION

ACTION SR03_FaultHandler:
tonFaultHandler(IN:=glb_bDevice1AllOP AND  glb_bAllSafetyOk, PT:= T#2S, Q=> , ET=> );
//停机故障信息(0,1 安全类报警)(2,3通讯类报警), (4,5,6,7伺服类报警)(8,9,10,11变频器类报警)
//(12,13,14,15气缸类报警)(16,17,18,19传感器类报警)(20,21,22,23真空类报警)(24...其它类报警) 
HMI_StopEvent[0].ID[1]:= NOT glb_bDevice1AllOP;//数粒Ethercat报警
HMI_StopEvent[0].ID[2]:= FALSE;//装罐Ethercat报警
HMI_StopEvent[0].ID[3]:= NOT glb_arSafeRelayNo_UN01[1];//安全继电器吸合报警		
HMI_StopEvent[0].ID[5]:= FALSE;	//机器人报警
HMI_StopEvent[0].ID[6]:= FALSE;//喷码机报警
HMI_StopEvent[0].ID[7]:= glb_MembraneAlarm;//

FOR iHmiErr:=1 TO 8 DO
	HMI_StopEvent[5].ID[iHmiErr]:=arHeat_AOI[iHmiErr].Error; //加热1—-8温度报警
END_FOR  

IF tonFaultHandler .Q THEN	
    HMI_StopEvent[0].ID[4]:= FALSE;			
    HMI_StopEvent[0].ID[8]:= NOT glb_bAirFeedback_UN01[1];//数粒系统气压异常报警
    HMI_StopEvent[0].ID[9]:= NOT glb_bAirFeedback_UN01[2];//装罐系统气压异常报警
    HMI_StopEvent[0].ID[10]:= arDropBufferCyclinder[1].o.Error;
	HMI_StopEvent[0].ID[11]:= arDropBufferCyclinder[2].o.Error;
	
	FOR iHmiErr:=1 TO 64 DO//伺服报警
	   HMI_StopEvent[1].ID[iHmiErr]:=arRealAxisAdmin[iHmiErr].o.Error OR (arErrorCodeDrive[iHmiErr]<>0);
	END_FOR
	
	FOR iHmiErr:=1 TO 40 DO//落料气缸报警
		HMI_StopEvent[2].ID[iHmiErr]:=arDropCylinder[iHmiErr].o.Error;
	END_FOR
	
	FOR iHmiErr:=1 TO 50 DO//气缸报警
		HMI_StopEvent[3].ID[iHmiErr]:=arPackCylinder[iHmiErr].o.Error;
	END_FOR
	
	FOR iHmiErr:=1 TO 40 DO//真空报警
		HMI_StopEvent[4].ID[iHmiErr]:=arPackVacuum[iHmiErr].o.Error;
	END_FOR
	
	FOR iHmiErr:=1 TO 40 DO//数粒报警
		HMI_StopEvent[6].ID[iHmiErr]:=arCounters[iHmiErr].Error;
	END_FOR
			
	FOR iHmiErr:=1 TO 40 DO//安全门报警
		HMI_GeneralEvent[1].ID[iHmiErr]:= arSafeDoorSts[iHmiErr];
	END_FOR    
	FOR iHmiErr:=1 TO 40 DO
	    HMI_GeneralEvent[2].ID[iHmiErr]:= arCounters[iHmiErr].Warning ;// 暂时屏蔽
    END_FOR  
END_IF

tongeneralEvent0[1](IN:=NOT arPackSensor[1].o.Value OR NOT arPackSensor[2].o.Value 
OR NOT arPackSensor[3].o.Value OR NOT arPackSensor[4].o.Value 
OR NOT arPackSensor[5].o.Value OR NOT arPackSensor[6].o.Value OR NOT arPackSensor[7].o.Value , 
PT:=T#3S , Q=> , ET=> );

HMI_GeneralEvent[0].ID[1]:=tongeneralEvent0[1].Q; //铝杯工位1缺料

tongeneralEvent0[2](IN:=NOT arPackSensor[8].o.Value OR NOT arPackSensor[9].o.Value 
OR NOT arPackSensor[10].o.Value OR NOT arPackSensor[11].o.Value 
OR NOT arPackSensor[12].o.Value OR NOT arPackSensor[13].o.Value OR NOT arPackSensor[14].o.Value , 
PT:=T#3S , Q=> , ET=> );

HMI_GeneralEvent[0].ID[2]:=tongeneralEvent0[2].Q ; //铝杯工位2缺料

tongeneralEvent0[3](IN:=NOT arPackSensor[22].o.Value	 , 
PT:=T#10S , Q=> , ET=> );  
HMI_GeneralEvent[0].ID[3]:=NOT HMI_PrinterConnected; //打印机未启用
HMI_GeneralEvent[0].ID[4]:=HMI_PrinterFault; //打印机未启用
tongeneralEvent0[4](IN:= arPackCylinder[22].i.InSensor AND NOT arPackSensor[20].o.Value 
AND (arPackMotor[3].Backward OR	arPackMotor[3].Forward) , 
PT:=T#10S , Q=> , ET=> );  



//////////////////////////////////////////////////////////////////////////////////
//////////////**********************************************************//////////
//////////////**********************************************************//////////
//////////////**********************************************************//////////
//////////////**********************************************************//////////
//////////////////////////////////////////////////////////////////////////////////
IF tonFaultHandler .Q THEN	
   		 
	FOR i:=1 TO 20 DO
		StopEvent[1].ID[i]:=arRealAxisAdmin[i].o.Error;//数粒伺服1-20报警
	END_FOR	
	FOR i:=1 TO 20 DO
		StopEvent[2].ID[i]:=arDropCylinder[i].o.Error;//数粒气缸21-40报警
	END_FOR

	FOR i:=21 TO 40 DO
		StopEvent[3].ID[i]:=arRealAxisAdmin[i].o.Error;//数粒伺服1-20报警
	END_FOR	
		 StopEvent[3].ID[40]:=FALSE;
	FOR i:=21 TO 40 DO
		StopEvent[4].ID[i]:=arDropCylinder[i].o.Error;//数粒气缸21-40报警
	END_FOR
         
	FOR i:=41 TO 48 DO //后段设备被取消 48台伺服 20210420
		StopEvent[5].ID[i]:=arRealAxisAdmin[i].o.Error; //伺服41-47报警  48报警
	END_FOR	
	FOR i:=1 TO 20 DO
		StopEvent[6].ID[i]:=arPackCylinder[i].o.Error;
	END_FOR
        StopEvent[6].ID[41]:=arPackCylinder[41].o.Error;
		
	FOR i:=1 TO 20 DO
		StopEvent[7].ID[i]:=arPackVacuum[i].o.Error;
	END_FOR		
		 
	FOR i:=1 TO 8 DO
		StopEvent[8].ID[i]:=arHeat_AOI[i].Error;
	END_FOR					  
		 
END_IF
StopEvent[8].ID[20]:=HMI_StopEvent[5].ID[20];	 
StopEvent[8].ID[21]:=HMI_StopEvent[5].ID[21];	
StopEvent[8].ID[22]:=HMI_StopEvent[5].ID[22];	
StopEvent[8].ID[23]:=HMI_StopEvent[5].ID[23];	
StopEvent[8].ID[24]:=HMI_StopEvent[5].ID[24];	
StopEvent[8].ID[25]:=HMI_StopEvent[5].ID[25];	
StopEvent[8].ID[26]:=HMI_StopEvent[5].ID[26];	
		  
StopEvent[0].ID[1]:= NOT glb_bDevice1AllOP;
StopEvent[0].ID[2]:= glb_MembraneAlarm;
StopEvent[0].ID[3]:= NOT glb_arSafeRelayNo_UN01[1];	
StopEvent[0].ID[4]:= NOT glb_bAirFeedback_UN01[1];	
StopEvent[0].ID[5]:= NOT glb_bAirFeedback_UN01[2];	
StopEvent[0].ID[6]:= HMI_PrinterFault;
StopEvent[0].ID[7]:= arDropBufferCyclinder[1].o.Error;
StopEvent[0].ID[8]:= arDropBufferCyclinder[2].o.Error;
	 
diUnitStopEvent0:=MEMCMP(pBuf1:=ADR(StopEvent[0]) , pBuf2:=ADR(arEventEmpty) , n:=SIZEOF(arEventEmpty));
diSys1StopEvent1:=MEMCMP(pBuf1:=ADR(StopEvent[1]) , pBuf2:=ADR(arEventEmpty) , n:=SIZEOF(arEventEmpty));
diSys1StopEvent2:=MEMCMP(pBuf1:=ADR(StopEvent[2]) , pBuf2:=ADR(arEventEmpty) , n:=SIZEOF(arEventEmpty));	 
diSys2StopEvent1:=MEMCMP(pBuf1:=ADR(StopEvent[3]) , pBuf2:=ADR(arEventEmpty) , n:=SIZEOF(arEventEmpty));
diSys2StopEvent2:=MEMCMP(pBuf1:=ADR(StopEvent[4]) , pBuf2:=ADR(arEventEmpty) , n:=SIZEOF(arEventEmpty));		  
diSys3StopEvent1:=MEMCMP(pBuf1:=ADR(StopEvent[5]) , pBuf2:=ADR(arEventEmpty) , n:=SIZEOF(arEventEmpty));
diSys3StopEvent2:=MEMCMP(pBuf1:=ADR(StopEvent[6]) , pBuf2:=ADR(arEventEmpty) , n:=SIZEOF(arEventEmpty));			   
diSys3StopEvent3:=MEMCMP(pBuf1:=ADR(StopEvent[7]) , pBuf2:=ADR(arEventEmpty) , n:=SIZEOF(arEventEmpty));	
diSys3StopEvent4:=MEMCMP(pBuf1:=ADR(StopEvent[8]) , pBuf2:=ADR(arEventEmpty) , n:=SIZEOF(arEventEmpty));

IF diSys1StopEvent1=0 AND diSys1StopEvent2=0 THEN
   bSys1StopError:=FALSE;
ELSE
   bSys1StopError:=TRUE;	
END_IF
	
IF diSys2StopEvent1=0 AND diSys2StopEvent2=0 THEN
   bSys2StopError:=FALSE;
ELSE
   bSys2StopError:=TRUE;	
END_IF 
		  
IF 	 diSys3StopEvent1=0 AND diSys3StopEvent2=0 AND diSys3StopEvent3=0 AND diSys3StopEvent3=0 AND diSys3StopEvent4=0
AND diUnitStopEvent0=0 THEN		
    bSys3StopError:=FALSE;
ELSE
    bSys3StopError:=TRUE;	
END_IF
					
IF bSys1StopError OR bSys2StopError OR bSys3StopError THEN
   loc_bAnyStopError:=TRUE;
   ELSE
   loc_bAnyStopError:=FALSE; 
END_IF
END_ACTION

ACTION SR04_Parameter:
arVirtualAxisAdmin[1].i.Vel:=HMI_MasterVelo;

//数粒伺服
FOR i:=1 TO 40 DO 
	arRealAxisAdmin[i].i.Vel:=HMI_CountersVelo;
	arRealAxisAdmin[i].i.Acc:=HMI_CountersAcc;
	arRealAxisAdmin[i].i.Dec:=HMI_CountersDec;
	arRealAxisAdmin[i].i.Jerk:=HMI_CountersDec*100;
END_FOR
//皮带1
arRealAxisAdmin[41].i.Vel:=HMI_BeltVelo[1];
arRealAxisAdmin[41].i.Acc:=HMI_BeltAcc[1];
arRealAxisAdmin[41].i.Dec:=HMI_BeltDec[1];
arRealAxisAdmin[41].i.HomeOffset:=HMI_HomeOffsetBelt[1];
//皮带2
arRealAxisAdmin[42].i.Vel:=HMI_BeltVelo[2];
arRealAxisAdmin[42].i.Acc:=HMI_BeltAcc[2];
arRealAxisAdmin[42].i.Dec:=HMI_BeltDec[2];
arRealAxisAdmin[42].i.HomeOffset:=HMI_HomeOffsetBelt[2];
//皮带3
arRealAxisAdmin[43].i.Vel:=HMI_BeltVelo[3];
arRealAxisAdmin[43].i.Acc:=HMI_BeltAcc[3];
arRealAxisAdmin[43].i.Dec:=HMI_BeltDec[3];
arRealAxisAdmin[43].i.HomeOffset:=HMI_HomeOffsetBelt[3];
//皮带4 //皮带5

//皮带6
arRealAxisAdmin[46].i.Dist:=222.25;
arRealAxisAdmin[46].i.HomeOffset:=HMI_HomeOffsetBelt[6];
arRealAxisAdmin[46].i.Vel:=HMI_BeltVelo[6];
arRealAxisAdmin[46].i.Acc:=HMI_BeltVelo[6]*100;
arRealAxisAdmin[46].i.Dec:=HMI_BeltVelo[6]*100;
//拉膜伺服
arRealAxisAdmin[47].i.Pos:=HMI_PullerPara[1];
arRealAxisAdmin[47].i.Dist:=HMI_PullerPara[1];
arRealAxisAdmin[47].i.JogVel:=HMI_PullerPara[2];
arRealAxisAdmin[47].i.JogAcc:=HMI_PullerPara[3];
arRealAxisAdmin[47].i.JogDec:=HMI_PullerPara[3];
arRealAxisAdmin[47].i.Vel:=HMI_PullerPara[2];
arRealAxisAdmin[47].i.Acc:=HMI_PullerPara[3];
arRealAxisAdmin[47].i.Dec:=HMI_PullerPara[3];
//皮带7 
arRealAxisAdmin[48].i.Dist:=150;
arRealAxisAdmin[48].i.HomeOffset:=HMI_HomeOffsetBelt[7];
arRealAxisAdmin[48].i.Vel:=HMI_BeltVelo[7];
arRealAxisAdmin[48].i.Acc:=HMI_BeltVelo[7]*100;
arRealAxisAdmin[48].i.Dec:=HMI_BeltVelo[7]*100;
//推瓶伺服
END_ACTION

ACTION SR05_Manual:
IF (Ref_MachineStateModel.Sts_Stopped OR Ref_MachineStateModel.Sts_Held) AND NOT  glb_bModeSwitch_UN01 THEN

	FOR i:=1 TO 40 DO
      arDropCylinder[i].i.ActiveIn:=FALSE;
	  arDropCylinder[i].i.ActiveOut:=FALSE;
	END_FOR
	
	FOR i:= 1 TO 20 DO
		arPackCylinder[i].i.ActiveIn:=FALSE;
		arPackCylinder[i].i.ActiveOut:=FALSE;	
    END_FOR
	
	FOR i:= 1 TO 10 DO
		arPackVacuum[i].i.ActiveIn:=FALSE;	
    END_FOR	


    FOR i:= 1 TO 40 DO
		IF HMI_ClearCounter[i] THEN
		   arRealAxisAdmin[i].i.Enable:=TRUE;
		END_IF
	END_FOR

    FOR i:= 1 TO 50 DO
	    arRealAxisAdmin[i].i.Mode:=1;
	END_FOR
ELSE
	 FOR i:=1 TO 32 DO 
		 FOR j:=1 TO 8 DO
			 DO_[i,j].ON:=FALSE;
			 DO_[i,j].Off:=FALSE;					 
		 END_FOR
	 END_FOR
	 FOR i:=50 TO 57 DO 
		 FOR j:=1 TO 8 DO
			 DO_[i,j].on:=FALSE;
			 DO_[i,j].Off:=FALSE;
		 END_FOR
	 END_FOR
	 FOR i:=1 TO 37 DO 
		 FOR j:=1 TO 8 DO
			 Di_[i,j].on:=FALSE;
			 Di_[i,j].Off:=FALSE;
		 END_FOR
	 END_FOR	 
	 
     FOR i:= 1 TO 50 DO
	     arRealAxisAdmin[i].i.Mode:=0;
		 HMI_AxisView[i].MoveReal:=FALSE;
	 END_FOR
	 HMI_AutoCut:=FALSE;
	 HMI_CutCnt:=0;
END_IF

//手动防护位
HMI_ManualInhibit[0]:=NOT arPackCylinder[1].i.InSensor OR NOT arPackCylinder[2].i.InSensor OR NOT arPackCylinder[3].i.InSensor  
OR NOT arPackCylinder[4].i.InSensor OR NOT arPackCylinder[5].i.InSensor OR NOT arPackCylinder[6].i.InSensor 
OR NOT arPackCylinder[7].i.InSensor OR NOT arPackCylinder[12].i.InSensor OR NOT arPackCylinder[15].i.InSensor
OR NOT arPackCylinder[16].i.InSensor OR NOT arPackCylinder[17].i.InSensor 
OR NOT arPackCylinder[10].i.InSensor OR NOT arPackCylinder[11].i.InSensor OR NOT arPackCylinder[41].i.InSensor ;

HMI_ManualInhibit[1]:=  arDropBufferCyclinder[1].i.InSensor AND arDropBufferCyclinder[2].i.InSensor;

CASE iAutoCut OF 
	0: IF HMI_AutoCut AND arRealAxisAdmin[47].o.PowerOn AND arRealAxisAdmin[46].o.PowerOn AND NOT glb_bModeSwitch_UN01 
       AND HMI_CutCnt>0 THEN
		  iAutoCut:=1;
		  iCutCnt:=iCutCnt+1;
	   END_IF
	1: 
       HMI_AxisView[47].MoveReal:=TRUE;
	   iAutoCut:=2;
	2: 
       tonAutoCut(IN:= TRUE, PT:= T#3S, Q=> , ET=> ); 
	   IF tonAutoCut.Q THEN 
	       tonAutoCut(IN:= FALSE, PT:= T#3S, Q=> , ET=> ); 
           iAutoCut:=3;	   
	   END_IF

